(* CODESYS project XtsCore.library
   Version: 0.12.1.34
   Title: XtsCore
   Placeholder: XtsCore
   Company: Beckhoff Automation LLC

Project tree, tasks and I/O mapping:
  libraries: Core, * (Beckhoff Automation LLC); Tc2_Math, * (Beckhoff Automation GmbH); Tc2_MC2, * (Beckhoff Automation GmbH); Tc2_Standard, * (Beckhoff Automation GmbH); Tc2_System, * (Beckhoff Automation GmbH); Tc2_Utilities, * (Beckhoff Automation GmbH); Tc3_EventLogger, * (Beckhoff Automation GmbH); Tc3_McCollisionAvoidance, * (Beckhoff Automation GmbH); Tc3_McCoordinatedMotion, * (Beckhoff Automation GmbH); Tc3_Module, * (Beckhoff Automation GmbH); Tc3_XTS_Utility, * (Beckhoff Automation GmbH)
  _Internal/
    _Needs Sorting/
      global variables TE2000
      function block TE2000_Hmi [ST]: RefreshXtsModule, RefreshXtsMovers, RefreshXtsParts, RefreshXtsPositionTriggers, RefreshXtsStations, RefreshXtsZones, BuildHMI, ControlObject, CyclicLogic, FB_Init, VisitComponent, VisitModule
      global variables TE2000_HMI_Parameters
    Collections/
      Modules/
        ModuleCollection/
          Interfaces/
            interface I_ContainXtsModules: XtsModules
            interface I_XtsModuleCollection: Clear, Count, Create, GetById, GetByOtcid, IsEmpty
            interface I_XtsModuleEnumerator: Current, CurrentItem, MoveToNext, ResetIterator
            function block XtsModuleCollectionAdapter [ST]: AddItem, Clear, Count, Current, CurrentItem, FB_Init, IsEmpty, MoveToNext, RemoveItem, ResetIterator
          function block XtsModuleCollection [ST]: Clear, Count, Create, GetById, GetByOtcid, IsEmpty, Current, CurrentItem, MoveToNext, ResetIterator, Dispose, FB_Exit, AcceptPeeker, CheckModuleId, GetModuleInstance
      Movers/
        MoverCollection/
          Interfaces/
            interface I_XtsMoverCollection: AcceptMoverVisitor, AddItem, Clear, Count, IsEmpty, Remove
            interface I_XtsMoverEnumerator: Current, CurrentItem, MoveToNext, ResetIterator
            interface I_XtsMoverMap: Map
          function block XtsMoverCollection [ST]: Current, CurrentItem, MoveToNext, ResetIterator, AcceptMoverVisitor, AcceptPeeker, AddItem, Clear, Count, IsEmpty, Map, Remove
        MoverList/
          Interfaces/
            interface I_XtsMoverList: Contains, GetAtIndex, InsertAtIndex, RemoveAtIndex
          function block XtsMoverList [ST]: AcceptMoverVisitor, AddItem, Clear, Count, IsEmpty, Map, Remove, Current, CurrentItem, MoveToNext, ResetIterator, Contains, GetAtIndex, InsertAtIndex, Movers, RemoveAtIndex
        MoverQueue/
          Interfaces/
            interface I_XtsMoverQueue: Clear, Count, Dequeue, Enqueue, Peek
          function block XtsMoverQueue [ST]: Current, CurrentItem, Map, MoveToNext, ResetIterator, AcceptMoverVisitor, Clear, Count, Dequeue, Enqueue, Movers, Peek
          function block XtsMoverUniqueQueue [ST]: Enqueue
      Parts/
        PartCollection/
          Interfaces/
            interface I_ContainXtsParts: Parts
            interface I_XtsPartCollection: AddItem, Clear, Count, GetById, GetByOtcid, IsEmpty, Remove
            interface I_XtsPartEnumerator: Current, CurrentItem, MoveToNext, ResetIterator
          function block XtsPartCollection [ST]: Current, CurrentItem, MoveToNext, ResetIterator, AcceptPeeker, AddItem, Clear, Count, FB_Exit, GetById, GetByOtcid, IsEmpty, Remove
      PositionTriggers/
        PositionTriggerCollection/
          Interfaces/
            interface I_XtsPositionTriggerCollection: AddItem, Clear, Count, IsEmpty, Remove
            interface I_XtsPositionTriggerEnumerator: Current, CurrentItem, MoveToNext, ResetIterator
          function block XtsPositionTriggerCollection [ST]: Current, CurrentItem, MoveToNext, ResetIterator, AcceptPeeker, AcceptXtsPositionTriggerVisitor, AddItem, Clear, Count, IsEmpty, Remove
      Stations/
        StationCollection/
          Interfaces/
            interface I_XtsStationCollection: AddItem, Clear, Count, IsEmpty, Remove
            interface I_XtsStationEnumerator: Current, CurrentItem, MoveToNext, ResetIterator
          function block XtsStationCollection [ST]: Current, CurrentItem, MoveToNext, ResetIterator, AcceptPeeker, AcceptStationVisitor, AddItem, Clear, Count, IsEmpty, Remove
      Tracks/
        TrackCollection/
          Interfaces/
            interface I_XtsTrackCollection: Clear, Count, Create, GetById, GetByOtcid, IsEmpty
            interface I_XtsTrackEnumerator: Current, CurrentIndex, MoveToNext, ResetIterator
          function block XtsTrackCollection [ST]: Clear, Count, Create, GetById, GetByOtcid, IsEmpty, Current, CurrentIndex, MoveToNext, ResetIterator, CheckTrackId, GetTrackInstance, FB_Exit
      Zones/
        ZoneCollection/
          Interfaces/
            interface I_XtsZoneCollection: AddItem, Clear, Count, IsEmpty, Remove
            interface I_XtsZoneEnumerator: Current, CurrentItem, MoveToNext, ResetIterator
          function block XtsZoneCollection [ST]: Current, CurrentItem, MoveToNext, ResetIterator, AcceptPeeker, AddItem, Clear, Count, IsEmpty, Remove
      interface I_ContainXtsMoverEnumerator: Movers
      interface I_ContainXtsMoverList: Movers
      interface I_OperatesOnMovers: Movers
    Frames/
      Interfaces/
        interface I_BaseFrame: FrameName
        interface I_FrameModulo: ModuloLength
        interface I_FrameOffset: OffsetToParent
        interface I_HasAReferenceFrame: ReferenceFrame, SetReferenceFrame
        interface I_InGlobalSpace: OffsetToGlobal
        interface I_Positionable: Position
        interface I_ReferencedPosition
        interface I_ReferenceFrame
      function block ReferencedPosition [ST]: Position, ReferenceFrame, SetReferenceFrame
      function block ReferenceFrame [ST]: FB_Init, FrameName, ModuloLength, OffsetToGlobal, OffsetToParent, ReferenceFrame, SetReferenceFrame
    GroupController/
      DUTs/
        data type E_MoverGroupState
      Interfaces/
        interface I_ContainXtsMoverGroupController: XtsMoverGroupController
        interface I_XtsMoverGroupController: AxesGroup, GroupStatus
      function block XtsGroupController [ST]: Disable, Enable, Reset, Accept, AxesGroup, Busy, CyclicLogic, DeregisterWithParent, Done, Enabled, Error, ErrorId, GroupStatus, RegisterWithParent, TaskName
    Module/
      Interfaces/
    Mover/
      MoverTaskBase/
        Interfaces/
          interface I_XtsMoverTask: Axis, Execute
          interface I_XtsMoverTaskCollection: AddTask, ErrorTask, GetTaskById, GetTaskByName, RemoveTaskById, RemoveTaskByInstance
          interface I_XtsMoverTaskResult: Aborted, CommandExecuted, TaskId
        function block XtsMoverTaskCollection [ST]: Busy, Error, ErrorId, ErrorTask, AddTask, CyclicLogic, FB_Init, GetTaskById, GetTaskByName, RemoveTaskById, RemoveTaskByInstance, Reset
        function block XtsMoverTaskResult [ST]: Aborted, CommandExecuted, CyclicLogic, Mover, TaskId
      Parameters/
        Interfaces/
          interface I_BaseDynamics: Acceleration, Deceleration, Direction, Jerk, Velocity
          interface I_CollisionAvoidanceDynamics: Gap
          interface I_CollisionAvoidanceGroupable: AxesGroup, IdentInGroup
          interface I_ContainSyncAxisParameters: SyncAxis
          interface I_HasXtsParameters: Parameters
          interface I_MoveToPositionParameters: Position
          interface I_MoveToStationParameters: Station
          interface I_SyncAxisParameters: MasterAxis, MasterStartDistance, MasterSyncPosition, Options_CA, RatioDenominator, RatioNumerator, SlaveSyncPosition, SyncMode, SyncStrategy
          interface I_XtsParameterSet: CopyFrom, CopyTo
          interface I_XtsTrackParameter: Track
        function block BaseDynamics [ST]: Acceleration, Deceleration, Direction, Jerk, Velocity
        function block CollisionAvoidanceDynamics [ST]: Gap
        function block MoveToPositionParameters [ST]: Position
        function block MoveToStationParameters [ST]: Station
        function block SyncAxisParameters [ST]: MasterAxis, MasterStartDistance, MasterSyncPosition, Options_CA, RatioDenominator, RatioNumerator, SlaveSyncPosition, SyncMode, SyncStrategy
        function block XtsParameterSet [ST]: Acceleration, CopyFrom, CopyTo, Deceleration, Direction, Gap, Jerk, Position, SyncAxis, Track, Velocity
        function block XtsTrackParameter [ST]: Track
      Properties/
        interface I_AxisTrackPositionable: Axis, MoverUtility, PartPosition, Position, TrackPosition
        function block PositionableBehavior [ST]: Axis, CyclicLogic, FB_Init, MoverUtility, PartPosition, Position, TrackPosition
      Status/
        Interfaces/
          interface I_ContainXtsMoverStatus: Status
          interface I_XtsMoverStatus: ActualAcceleration, ActualVelocity, AvoidingCollision, Axis, CommandedPosition, CommandedStation, CurrentTrack, IdentInGroup, InSync, MoverInGroup, SetAcceleration, SetVelocity
        function block XtsMoverStatus [ST]: ActualAcceleration, ActualVelocity, AvoidingCollision, Axis, CommandedPosition, CommandedStation, CurrentTrack, FB_Init, IdentInGroup, InSync, MoverInGroup, SetAcceleration, SetVelocity
      Tasks/
        Interfaces/
          interface I_AxesGroupTask
          interface I_AxisRef: Axis
          interface I_EnableXtsMoverTask: Disable, Disabled, Enable, Enabled, InhibitFeedBackward, InhibitFeedForward, Override
          interface I_MoveToStationTask
          interface I_TakesTrackId: TrackId
        Wrappers/
          Interfaces/
            interface I_ActivateTrack: Execute, TrackId, Busy, Error, ErrorId
            interface I_AxisOnGroup: Execute, IdentInGroup, Busy, Error, ErrorId
            interface I_BaseCollisionAvoidance: Execute, Gap, Active, Busy, Error, ErrorId
            interface I_DynamicsCollisionAvoidance: Acceleration, Deceleration, Jerk, Velocity, CommandAborted
            interface I_GearInPosCA: BufferMode, ContinuousUpdate, MasterStartDistance, MasterSyncPosition, Options, RatioDenominator, RatioNumerator, SlaveSyncPosition, SyncMode, SyncStrategy, InSync, StartSync
            interface I_HaltCa: Deceleration, Jerk, Options, CommandAborted
            interface I_MoveToPositionCA: BufferMode, ContinuousUpdate, Direction, Options, Position, CommandAborted
            interface I_Power: BufferMode, Enable, Enable_Negative, Enable_Positive, Options, Override, Busy, Error, ErrorId, Status
            interface I_ResetAxis: Execute, Busy, Error, ErrorId
          function block ActivateTrack [ST]: Execute, TrackId, Busy, Done, Error, ErrorId
          function block AddAxisToGroup [ST]: Execute, IdentInGroup, Busy, Done, Error, ErrorId
          function block GearInPosCa [ST]: Acceleration, BufferMode, ContinuousUpdate, Deceleration, Execute, Gap, Jerk, MasterStartDistance, MasterSyncPosition, Options, RatioDenominator, RatioNumerator, SlaveSyncPosition, SyncMode, SyncStrategy, Velocity, Active, Busy, CommandAborted, Done, Error, ErrorId, InSync, StartSync
          function block HaltCa [ST]: Deceleration, Execute, Gap, Jerk, Options, Active, Busy, CommandAborted, Done, Error, ErrorId
          function block MoveToAbsolutePositionCA [ST]: Acceleration, BufferMode, ContinuousUpdate, Deceleration, Direction, Execute, Gap, Jerk, Options, Position, Velocity, Active, Busy, CommandAborted, Done, Error, ErrorId
          function block MoveToRelativePositionCA [ST]: Acceleration, BufferMode, ContinuousUpdate, Deceleration, Direction, Execute, Gap, Jerk, Options, Position, Velocity, Active, Busy, CommandAborted, Done, Error, ErrorId
          function block PowerAxis [ST]: BufferMode, Enable, Enable_Negative, Enable_Positive, Options, Override, Busy, Error, ErrorId, Status
          function block RemoveAxisFromGroup [ST]: Execute, IdentInGroup, Busy, Done, Error, ErrorId
          function block ResetMover [ST]: Execute, Busy, Done, Error, ErrorId
        function block _DefaultMoverTasks [ST]
        function block _MoverTasks [ST]: ActivateTrack, AddToGroup, EnableAxis, HaltMover, MoveRelative, MoveToPosition, MoveToStation, MoveVelocity, RemoveFromGroup, ResetAxis, ResetToDefault, SyncToAxis
        function block ActivateTrackTask [ST]: Axis, CyclicLogic, Execute, FB_Init, Reset, TrackId
        function block AddToGroupTask [ST]: AxesGroup, Axis, CyclicLogic, Execute, FB_Init, IdentInGroup, Reset
        function block EnableAxisTask [ST]: Axis, CyclicLogic, Disable, Disabled, Enable, Enabled, Execute, FB_Init, InhibitFeedBackward, InhibitFeedForward, Override, Reset
        function block HaltMoverCATask [ST]: Axis, CyclicLogic, Execute, FB_Init, Interrupted, Reset
        function block MoveRelativeCATask [ST]: Axis, CyclicLogic, Execute, FB_Init, Reset
        data type MoverTaskID
        function block MoveToPositionCATask [ST]: Axis, CyclicLogic, Execute, FB_Init, Reset
        function block MoveToStationTask [ST]: Axis, CyclicLogic, Execute, FB_Init, Reset, Station
        function block MoveVelocityTask [ST]: Axis, CyclicLogic, Execute, FB_Init, Reset
        function block RemoveFromGroupTask [ST]: AxesGroup, Axis, CyclicLogic, Execute, FB_Init, IdentInGroup, Reset
        function block ResetAxisTask [ST]: Axis, CyclicLogic, Execute, FB_Init, Reset
        function block SyncToAxisTask [ST]: Axis, CyclicLogic, Execute, FB_Init, Reset
    NullObjects/
      function GetSeverityString [ST]
      interface I_NullObject
      function block NullAxisRef [ST]: Axis
      function block NullMechatronicsLocalLog [ST]: Clear, Commands, DetailedCommands
      function block NullMechatronicsLogger [ST]: LogMessage, LogMessageInstance
      function block NullMechatronicsTracePublisher [ST]: LogMessage, LogMessageInstance, Subscribe, Unsubscribe
      function block NullMoverCollection [ST]: AcceptMoverVisitor, AddItem, Clear, Count, Current, CurrentItem, IsEmpty, Map, MoveToNext, Remove, ResetIterator
      global variables NullObjects
      function block NullPositionTriggerCollection [ST]: AcceptXtsPositionTriggerVisitor, AddItem, Clear, Count, Current, CurrentItem, IsEmpty, MoveToNext, Remove, ResetIterator
      function block NullReferenceFrame [ST]: FrameName, ModuloLength, OffsetToGlobal, OffsetToParent, ReferenceFrame, SetReferenceFrame
      function block NullStation [ST]: AcceptStationVisitor, CommandLog, CyclicLogic, DeregisterMover, Disable, Enable, Enabled, GetMover, IsMoverRegistered, MoverIsPresent, Movers, Position, RegisterMover, Status, TracePublisher
      function block NullStationCollection [ST]: AcceptStationVisitor, AddItem, Clear, Count, Current, CurrentItem, IsEmpty, MoveToNext, Remove, ResetIterator
      function block NullSyncAxisParameters [ST]: MasterAxis, MasterStartDistance, MasterSyncPosition, Options_CA, RatioDenominator, RatioNumerator, SlaveSyncPosition, SyncMode, SyncStrategy
      function block NullXtsModule [ST]: Accept, AcceptXtsModuleVisitor, CurveAngle, CyclicLogic, Dispose, Gap, HMI, Id, Initialize, Initialized, Length, Module24Vdc, Module48Vdc, ModuleReady, Name, Otcid, RegisterWithParent, Utility, Vdc24Okay, Vdc48Okay, XtsModuleType
      function block NullXtsModuleCollection [ST]: Clear, Count, Create, Current, CurrentItem, Dispose, GetById, GetByOtcid, IsEmpty, MoveToNext, ResetIterator
      function block NullXtsMover [ST]: Accept, AcceptMoverVisitor, ActivateTrack, AddToGroup, Axis, Busy, CommandLog, CurrentTask, DeregisterWithParent, Disable, Enable, Enabled, Error, ErrorId, Halt, Initialize, Initialized, InPosition, InVelocity, LastCyclePosition, ManualGroupControl, MoverData, MoveRelative, MoverId, MoverTasks, MoverUtility, MoveToPosition, MoveToPositionRelative, MoveToStation, MoveVelocity, Name, Parameters, Position, RefreshMoverId, RegisterWithParent, RemoveFromGroup, Reset, Status, SyncToAxis, SyncToMover, TracePublisher, Tracks, VirtualMover
      function block NullXtsMoverData [ST]
      function block NullXtsMoverList [ST]: AcceptMoverVisitor, AddItem, Clear, Contains, Count, Current, CurrentItem, GetAtIndex, InsertAtIndex, IsEmpty, Map, Mover, MoveToNext, Remove, RemoveAtIndex, ResetIterator
      function block NullXtsMoverStatus [ST]: ActualAcceleration, ActualVelocity, AvoidingCollision, Axis, CommandedPosition, CommandedStation, CurrentStation, CurrentTrack, IdentInGroup, InSync, MoverInGroup, SetAcceleration, SetVelocity
      function block NullXtsMoverTask [ST]: Axis, CyclicLogic, Execute, Reset, TaskId, TaskName
      function block NullXtsMoverTaskCollection [ST]: AddTask, ErrorTask, GetTaskById, GetTaskByName, RemoveTaskById, RemoveTaskByInstance
      function block NullXtsMoverTaskResult [ST]: Aborted, Busy, CommandExecuted, Error, ErrorId, TaskId, TaskName
      function block NullXtsParameterSet [ST]: Acceleration, CopyFrom, CopyTo, Deceleration, Direction, Gap, Jerk, Position, SyncAxis, Track, Velocity
      function block NullXtsPart [ST]: Accept, AcceptXtsModuleVisitor, AcceptXtsPartVisitor, Components, CyclicLogic, DeregisterComponent, DeregisterCyclic, DeregisterInitialize, DeregisterModule, DeregisterWithParent, Dispose, Id, Initialize, Initialized, Modules, Name, NumberModulesNotReady, NumberModulesReady, PartReady, Properties, RegisterComponent, RegisterCyclic, RegisterInitialize, RegisterModule, RegisterWithParent, ResetComponents, ResetModules, Utility, Vdc24Okay, Vdc48Okay, XtsModules, XtsPartId
      function block NullXtsPartCollection [ST]: AddItem, Clear, Count, Current, CurrentItem, GetById, GetByOtcid, IsEmpty, MoveToNext, Remove, ResetIterator
      function block NullXtsPartTask [ST]: Busy, Error, ErrorId, TaskName, XtsPartId
      function block NullXtsPositionTrigger [ST]: Accept, AcceptXtsPositionTriggerVisitor, CommandLog, DeregisterMover, DeregisterWithParent, Disable, Enable, Enabled, GetMover, IsMoverRegistered, MoverIsPresent, MoverQueue, Movers, Name, Position, RegisterMover, RegisterWithParent, Status, TracePublisher
      function block NullXtsPositionTriggerStatus [ST]: NumberOfMoverEvents, NumberOfMoversRegistered
      function block NullXtsStationStatus [ST]: CurrentMoverId, CurrentMoverName, NumberOfMoversRegistered
      function block NullXtsSystem [ST]: Accept, AcceptMoverVisitor, AcceptStationVisitor, AcceptXtsModuleVisitor, AcceptXtsPartVisitor, AcceptXtsPositionTriggerVisitor, AcceptXtsZoneVisitor, AxesGroupRef, Busy, CAGroupErrorId, CaGroupStatus, CommandLog, Components, Config, CurrentTask, CyclicLogic, DeregisterComponent, DeregisterCyclic, DeregisterInitialize, DeregisterModule, DeregisterWithParent, Disable, DisableGroup, DisableMovers, Enable, Enabled, EnableGroup, EnableMovers, Environment, Error, ErrorId, Initialize, Initialized, ManualDiagnoser, Modules, Movers, MoversEnabled, Name, Parameters, Parts, PositionTriggers, RegisterComponent, RegisterCyclic, RegisterInitialize, RegisterModule, RegisterWithParent, Reset, ResetCaGroup, ResetComponents, ResetModules, ResetMovers, RetriggerMoverDetection, Stations, Status, TracePublisher, Tracks, TriggerMoverDetection, TriggerMoverIdentification, Utility, UtilityProperties, XpuId, XtsTasks, Zones
      function block NullXtsSystemConfiguration [ST]: CommandPositionTriggersOnDisable, CommandPositionTriggersOnEnable, CommandStationsOnDisable, CommandStationsOnEnable
      function block NullXtsSystemStatus [ST]: CyclicLogic, NumberOfMovers, NumberOfParts, NumberOfPositionTriggers, NumberOfStations, NumberOfTracks, NumberOfZones, NumberPartsNotReady, NumberPartsReady, Simulated, Vdc24Okay, Vdc48Okay
      function block NullXtsSystemTasks [ST]: AddTask, CyclicLogic, GetTaskById, GetTaskByName, RemoveTaskById, RemoveTaskByInstance
      function block NullXtsTask [ST]: Busy, Error, ErrorId, TaskId, TaskName, XpuId
      function block NullXtsTrack [ST]: Dispose, Id, Length, Offset, Otcid, Polarity, Utility
      function block NullXtsTrackCollection [ST]: Clear, Count, Create, Current, CurrentIndex, GetById, GetByOtcid, IsEmpty, MoveToNext, ResetIterator
      function block NullXtsZone [ST]: Accept, AcceptMoverVisitor, AcceptXtsZoneVisitor, CommandLog, DeregisterWithParent, EndPosition, GetSortedMover, IsMoverInZone, Length, MonitoredMovers, Movers, Name, RegisterWithParent, StartPosition, Status, TracePublisher
      function block NullXtsZoneStatus [ST]: NumberOfMoversInZone
      function block NullZoneCollection [ST]: AddItem, Clear, Count, Current, CurrentItem, IsEmpty, MoveToNext, Remove, ResetIterator
    Parts/
      Properties/
        interface I_ContainXtsPartProperties: Properties
        interface I_XtsPartProperties: General
        interface I_XtsPartPropertiesGeneral: ModuleSide, Offset, OTCID
        function block XtsPartProperties [ST]: General
        function block XtsPartPropertiesGeneral [ST]: ModuleSide, Offset, OTCID
      Tasks/
        Interfaces/
          interface I_XtsPartInitializeTask
          interface I_XtsPartTask: XtsPartId
          interface I_XtsPartTaskResult
        function block InitializeXtsPartTask [ST]: Initialize, Initialized, XtsPartId
      interface I_XtsPartId: XtsPartId
    Peeker/
      Interfaces/
        interface I_XtsModuleCollectionPeeker: SetCollection
        interface I_XtsMoverCollectionPeeker: SetCollection
        interface I_XtsPartCollectionPeeker: SetCollection
        interface I_XtsPositionTriggerCollectionPeeker: SetCollection
        interface I_XtsStationCollectionPeeker: SetCollection
        interface I_XtsZoneCollectionPeeker: SetCollection
    PositionTrigger/
      Status/
        Interfaces/
          interface I_ContainXtsPositionTriggerStatus: Status
          interface I_XtsPositionTriggerStatus: NumberOfMoverEvents, NumberOfMoversRegistered
        function block XtsPositionTriggerStatus [ST]: FB_Init, NumberOfMoverEvents, NumberOfMoversRegistered, SetRegisteredMovers
    Station/
      DUT/
        data type E_ThresholdEvent
      Interfaces/
        interface I_MoverMonitor: GetMover, MonitoredMovers, MoverPresent
        interface I_StationTaskCollection
      Status/
        Interfaces/
          interface I_ContainXtsStationStatus: Status
          interface I_XtsStationStatus: NumberOfMoversRegistered
        function block XtsStationStatus [ST]: FB_Init, NumberOfMoversRegistered, SetRegisteredMovers
      function CheckForThresholdEvent [ST]
      function block MoverMonitorTask [ST]: CyclicLogic, FB_Init, GetMover, MonitoredMovers, MoverPresent
      function block MoverThresholdMonitorTask [ST]: CyclicLogic, FB_Init, GetMover, MonitoredMovers, MoverPresent, SetMonitoredMovers
    TaskBase/
      Interfaces/
        interface I_TaskResult: TaskName
      function block BaseTaskResult [ST]: Busy, Error, ErrorId, TaskName
    Tracing/
      function block XtsCoreEventLogger [ST]: LogMessage, LogMessageInstance
    Tracks/
      Interfaces/
        interface I_XtsTrack: Id, Length, Offset, Otcid, Polarity, Utility
      function block XtsTrack [ST]: Dispose, Id, Length, Offset, Otcid, Polarity, Utility
    XtsSystem/
      Base/
        Interfaces/
          interface I_XtsTask: XpuId
          interface I_XtsTaskCollection: AddTask, GetTaskById, GetTaskByName, RemoveTaskById, RemoveTaskByInstance
          interface I_XtsTaskResult: TaskId
        function block XtsTaskCollection [ST]: AddTask, Busy, CyclicLogic, Error, ErrorId, FB_Init, GetTaskById, GetTaskByName, RemoveTaskById, RemoveTaskByInstance, Reset
        function block XtsTaskResult [ST]: TaskId
      Properties/
        Interfaces/
          interface I_ContainXtsSystemProperties: UtilityProperties
          interface I_XtsSystemUtilityProperties: Mover
          interface I_XtsSystemUtilityPropertiesMover: XtsMagnetPlateType, XtsMoverType
        function block XtsSystemConfiguration [ST]: CommandPositionTriggersOnDisable, CommandPositionTriggersOnEnable, CommandStationsOnDisable, CommandStationsOnEnable
        function block XtsSystemUtilityProperties [ST]: Mover
        function block XtsSystemUtilityPropertiesMover [ST]: XtsMagnetPlateType, XtsMoverType
      Status/
        Interfaces/
          interface I_ContainXtsSystemStatus: Status
          interface I_XtsSystemStatus: NumberOfMovers, NumberOfParts, NumberOfPositionTriggers, NumberOfStations, NumberOfTracks, NumberOfZones, NumberPartsNotReady, NumberPartsReady, Simulated, Vdc24Okay, Vdc48Okay
        function block XtsSystemStatus [ST]: CyclicLogic, FB_Init, NumberOfMovers, NumberOfParts, NumberOfPositionTriggers, NumberOfStations, NumberOfTracks, NumberOfZones, NumberPartsNotReady, NumberPartsReady, Simulated, Vdc24Okay, Vdc48Okay
      Tasks/
        Interfaces/
          interface I_XtsDisableTask: AxesGroup
          interface I_XtsEnableTask: AxesGroup
          interface I_XtsExecutableTask: Execute
          interface I_XtsInitializeTask
          interface I_XtsMoverDetectionTask
          interface I_XtsMoverIdentificationTask
          interface I_XtsMoverRedetectionTask
        function block _DefaultXtsTasks [ST]
        function block _XtsTasks [ST]: DisableXtsTask, EnableXtsTask, InitializeXtsTask, MoverDetectionTask, MoverIdentificationTask, MoverRedetectionTask
        function block DisableXtsTask [ST]: AxesGroup, CyclicLogic, Execute, FB_Init, Reset, XpuId, XtsMoverCommander, XtsMoverGroupController
        function block EnableXtsTask [ST]: AxesGroup, CyclicLogic, Execute, FB_Init, Reset, XpuId, XtsMoverCommander, XtsMoverGroupController
        function block InitializeXtsTask [ST]: Initialize, Initialized, InfoServerSetup, MoverSetup, PartSetup, TrackSetup, FB_Init, Reset, XpuId
        function block MoverDetectionTask [ST]: Execute, FB_Init, XpuId
        function block MoverIdentificationTask [ST]: CyclicLogic, Execute, FB_Init, Reset, XpuId
        function block MoverRedetectionTask [ST]: Execute, FB_Init, XpuId
        data type XtsSystemTaskId
      function block ManualDebugger [ST]: PartIdForModules, RefreshCollections, SetCollections
    Zone/
      Interfaces/
        interface I_MoverInPositionChecker: IsMoverInPosition
        interface I_XtsMoverComparer: Compare
        interface I_ZoneMonitor
      Properties/
        Interfaces/
          interface I_SingleDimensionZone: EndPosition, StartPosition
        function block _DefaultZoneProperties [ST]
        function block _DefaultZonePropertyBackers [ST]: SingleDimensionBacker
        function block SingleDimensionZone [ST]: EndPosition, StartPosition
      Status/
        Interfaces/
          interface I_ContainXtsZoneStatus: Status
          interface I_XtsZoneStatus: NumberOfMoversInZone
        function block XtsZoneStatus [ST]: FB_Init, NumberOfMoversInZone, SetMoverCollection
      function MoverDistance [ST]
      function block MoverZoneDistanceComparer [ST]: Compare, FB_Init
      function block SingleDimensionChecker [ST]: FB_Init, IsMoverInPosition
      function block ZoneMonitor [ST]: CyclicLogic, FB_Init, MonitoredMovers, Movers
    data type E_XtsLogMessage
  HMI/
    DUT/
      data type ST_LocalLogbook_HMI
      data type ST_MoverCommands_HMI
      data type ST_XtsModule_HMI
      data type ST_XtsMover_HMI
      data type ST_XtsMover_Parameters_HMI
      data type ST_XtsPart_HMI
      data type ST_XtsPartHmiHelper
      data type ST_XtsPositionTrigger_HMI
      data type ST_XtsStation_HMI
      data type ST_XtsSystem_HMI
      data type ST_XtsTrack_HMI
      data type ST_XtsZone_HMI
    function block XtsBasicHmi [ST]: FB_Init, Accept, BuildHMI, ControlObject, CyclicLogic, VisitComponent, VisitModule
    function block XtsModule_HMI [ST]: ControlObject, CyclicLogic, FB_Init, XtsModule
    function block XtsMover_HMI [ST]: ControlObject, CyclicLogic, FB_Init, XtsMover
    function block XtsPart_HMI [ST]: ControlObject, CyclicLogic, FB_Init, XtsPart
    function block XtsPositionTrigger_HMI [ST]: ControlObject, CyclicLogic, FB_Init, XtsPositionTrigger
    function block XtsStation_HMI [ST]: ControlObject, CyclicLogic, FB_Init, XtsStation
    function block XtsSystem_HMI [ST]: ControlObject, CyclicLogic, FB_Init
    function block XtsZone_HMI [ST]: ControlObject, CyclicLogic, FB_Init
  Logging/
    Interfaces/
      interface I_ContainXtsLocalLog: CommandLog
      interface I_ContainXtsTracePublisher: TracePublisher
      interface I_XtsLocalLog: Clear, Commands, DetailedCommands
      interface I_XtsLocalLogger
      interface I_XtsLogCommand
      interface I_XtsLogger
      interface I_XtsTracePublisher: Subscribe, Unsubscribe
    function block XtsLocalLogger [ST]: Clear, Commands, DetailedCommands, FB_Init, LogMessage, LogMessageInstance
    function block XtsLogCommand [ST]: Arguments, Message, MessageId, Severity, SourceId, SourceName, TimeStamp
    function block XtsTracePublisher [ST]: LogMessage, LogMessageInstance, Subscribe, Unsubscribe
  MoverVisitors/
    Interfaces/
      interface I_XtsMoverVisitorTask: ExecuteOn
    MoverCollectionVisitors/
    function block XtsMoverActivateTrack [ST]: CopyParametersFrom, TrackId, XtsMoverVisitee, Aborted, Busy, CommandExecuted, Error, ErrorId, ExecuteOn, TaskId, TaskName, VisitMover
    function block XtsMoverAddToGroup [ST]: AxesGroup, IdentInGroup, XtsMoverVisitee, Aborted, Busy, CommandExecuted, Error, ErrorId, ExecuteOn, TaskId, TaskName, VisitMover
    function block XtsMoverDisabler [ST]: XtsMoverVisitee, Aborted, Busy, CommandExecuted, Error, ErrorId, ExecuteOn, TaskId, TaskName, VisitMover
    function block XtsMoverEnabler [ST]: XtsMoverVisitee, Aborted, Busy, CommandExecuted, Error, ErrorId, ExecuteOn, TaskId, TaskName, VisitMover
    function block XtsMoverHalt [ST]: CopyParametersFrom, Deceleration, Gap, Jerk, XtsMoverVisitee, Aborted, Busy, CommandExecuted, Error, ErrorId, ExecuteOn, TaskId, TaskName, VisitMover
    function block XtsMoverMoveToPosition [ST]: Acceleration, CopyParametersFrom, Deceleration, Direction, Gap, Jerk, Position, Velocity, XtsMoverVisitee, Aborted, Busy, CommandExecuted, Error, ErrorId, ExecuteOn, TaskId, TaskName, VisitMover
    function block XtsMoverMoveToStation [ST]: Acceleration, CopyParametersFrom, Deceleration, Direction, Gap, Jerk, Station, Velocity, XtsMoverVisitee, Aborted, Busy, CommandExecuted, Error, ErrorId, ExecuteOn, TaskId, TaskName, VisitMover
    function block XtsMoverMoveVelocity [ST]: Acceleration, CopyParametersFrom, Deceleration, Direction, Gap, Jerk, Velocity, XtsMoverVisitee, Aborted, Busy, CommandExecuted, Error, ErrorId, ExecuteOn, TaskId, TaskName, VisitMover
    function block XtsMoverRemoveFromGroup [ST]: AxesGroup, IdentInGroup, XtsMoverVisitee, Aborted, Busy, CommandExecuted, Error, ErrorId, ExecuteOn, TaskId, TaskName, VisitMover
  Project Information/
    function F_GetCompany [ST]
    function F_GetTitle [ST]
    function F_GetVersion [ST]
  Utilities/
    Logging/
      global variables XtsTrace
    Validators/
      function block AllMoversValidator [ST]: Valid
      function block NoMoversValidator [ST]: Valid
    function IsNullObject [ST]
    function IsValidObject [ST]
  Version/
    global variables Global_Version
  XtsModule/
    Interfaces/
      interface I_AcceptXtsModuleVisitor: AcceptXtsModuleVisitor
      interface I_ContainXtsPartModuleUtility: Utility
      interface I_XtsModule: CurveAngle, Gap, Id, Length, ModuleReady, Otcid, Vdc24Okay, Vdc48Okay, XtsModuleType
      interface I_XtsModuleVisitor: VisitXtsModule
    function block XtsModule [ST]: DeregisterWithParent, RegisterWithParent, Dispose, Initialize, Initialized, CurveAngle, Gap, Id, Length, ModuleReady, Otcid, Utility, Vdc24Okay, Vdc48Okay, XtsModuleType, AcceptXtsModuleVisitor, CyclicLogic
  XtsMover/
    Interfaces/
      interface I_AcceptXtsMoverVisitors: AcceptMoverVisitor
      interface I_XtsCommands: ActivateTrack, AddToGroup, Halt, MoveRelative, MoveToPosition, MoveToStation, MoveVelocity, RemoveFromGroup, SyncToAxis, SyncToMover
      interface I_XtsMover: CurrentTask, InPosition, InVelocity, LastCyclePosition, ManualGroupControl, MoverId, MoverTasks, Position, RefreshMoverId, Tracks, VirtualMover
      interface I_XtsMoverUtility: MoverUtility
      interface I_XtsMoverValidator: Valid
      interface I_XtsMoverVisitor: VisitMover
    XtsMoverData/
      Interfaces/
        interface I_ContainXtsMoverData: MoverData
        interface I_XtsMoverData
    function block XtsMover [ST]: CyclicLogic, MoverTasks, MoverUtility, RefreshMoverId, RegisterWithParent, ActivateTrack, AddToGroup, Disable, Enable, Halt, MoveRelative, MoveToPosition, MoveToStation, MoveVelocity, RemoveFromGroup, Reset, SyncToAxis, SyncToMover, FB_Init, Initialize, Initialized, Axis, InhibitFeedBackward, InhibitFeedForward, InPosition, InVelocity, LastCyclePosition, ManualGroupControl, MoverData, MoverId, Override, Parameters, Position, Tracks, VirtualMover, Busy, CurrentTask, Enabled, Error, ErrorId, Status, CommandLog, TracePublisher, AcceptMoverVisitor
  XtsMoverCommander/
    Interfaces/
      interface I_ContainXtsMoverCommander: XtsMoverCommander
      interface I_XtsMoverCommander: ActivateTrack, AddToGroup, Disable, Enable, Halt, MoveToPosition, MoveToStation, MoveVelocity, RemoveFromGroup
    function block XtsMoverCommander [ST]: ActivateTrack, AddToGroup, Disable, Enable, Halt, MoveToPosition, MoveToStation, MoveVelocity, RemoveFromGroup, Busy, CurrentTask, Error, ErrorId, Parameters, TaskName
  XtsPart/
    Interfaces/
      interface I_AcceptXtsPartVisitor: AcceptXtsPartVisitor
      interface I_ContainXtsPartUtility: Utility
      interface I_XtsPart: PartReady, Vdc24Okay, Vdc48Okay
      interface I_XtsPartVisitor: VisitXtsPart
    function block XtsPart [ST]: FB_Init, Dispose, Initializing, Properties, PartReady, Vdc24Okay, Vdc48Okay, AcceptXtsModuleVisitor, AcceptXtsPartVisitor, OnCyclicCall, Utility, XtsModules, XtsPartId
  XtsPositionTrigger/
    Interfaces/
      interface I_AcceptXtsPositionTriggerVisitor: AcceptXtsPositionTriggerVisitor
      interface I_Queueable: MoverQueue
      interface I_VisitXtsPositionTrigger: VisitXtsPositionTrigger
      interface I_XtsPositionTrigger: Movers
    function block XtsPositionTrigger [ST]: FB_Init, Disable, Enable, Enabled, CommandLog, TracePublisher, AcceptXtsPositionTriggerVisitor, CyclicLogic, DeregisterMover, GetMover, IsMoverRegistered, MoverIsPresent, MoverQueue, Movers, Position, RegisterMover, Status
  XtsStation/
    Interfaces/
      interface I_AcceptXtsStationVisitor: AcceptStationVisitor
      interface I_MoverPositionMonitor
      interface I_Station: DeregisterMover, GetMover, IsMoverRegistered, MoverIsPresent, RegisterMover
      interface I_XtsStation
      interface I_XtsStationVisitor: VisitStation
    function block XtsStation [ST]: FB_Init, Disable, Enable, Enabled, CommandLog, TracePublisher, AcceptStationVisitor, CyclicLogic, DeregisterMover, GetMover, IsMoverRegistered, MoverIsPresent, Movers, Position, RegisterMover, Status
  XtsSystem/
    Interfaces/
      interface I_ContainXtsEnvironment: Environment
      interface I_ContainXtsMovers: Movers
      interface I_ContainXtsPositionTriggers: PositionTriggers
      interface I_ContainXtsStations: Stations
      interface I_ContainXtsTracks: Tracks
      interface I_ContainXtsUtility: Utility
      interface I_ContainXtsZones: Zones
      interface I_XtsSystem: AxesGroupRef, Busy, CAGroupErrorId, CaGroupStatus, Config, CurrentTask, Error, ErrorId, ManualDiagnoser, MoversEnabled, XtsTasks
      interface I_XtsSystemCommands: DisableGroup, DisableMovers, EnableGroup, EnableMovers, ResetCaGroup, ResetMovers, RetriggerMoverDetection, TriggerMoverDetection, TriggerMoverIdentification
      interface I_XtsSystemConfiguration: CommandPositionTriggersOnDisable, CommandPositionTriggersOnEnable, CommandStationsOnDisable, CommandStationsOnEnable
      interface I_XtsXpuId: XpuId
    function block XtsSystem [ST]: Movers, Parameters, Parts, PositionTriggers, Stations, Tracks, XtsTasks, Zones, Disable, DisableGroup, DisableMovers, Enable, EnableGroup, EnableMovers, Reset, ResetCaGroup, ResetMovers, RetriggerMoverDetection, TriggerMoverDetection, TriggerMoverIdentification, FB_Init, Initializing, UtilityProperties, AxesGroupRef, Busy, CAGroupErrorId, CaGroupStatus, Config, CurrentTask, Enabled, Environment, Error, ErrorId, MoversEnabled, Status, Utility, XpuId, CommandLog, TracePublisher, AcceptMoverVisitor, AcceptStationVisitor, AcceptXtsModuleVisitor, AcceptXtsPartVisitor, AcceptXtsPositionTriggerVisitor, AcceptXtsZoneVisitor, ManualDiagnoser, OnCyclicCall
  XtsZone/
    Interfaces/
      interface I_AcceptXtsZoneVisitor: AcceptXtsZoneVisitor
      interface I_MonitorsMovers: MonitoredMovers
      interface I_XtsZone: GetSortedMover, IsMoverInZone
      interface I_XtsZoneVisitor: VisitZone
    function block XtsZone [ST]: FB_Init, EndPosition, StartPosition, CommandLog, TracePublisher, AcceptMoverVisitor, AcceptXtsZoneVisitor, CyclicLogic, GetSortedMover, IsMoverInZone, MonitoredMovers, Movers, Status
  global variables XtsCoreParameters
*)

// _Internal/GroupController/DUTs/E_MoverGroupState
{attribute 'qualified_only'}
{attribute 'strict'}
{attribute 'to_string'}
TYPE E_MoverGroupState :
(
	Disabled := 0,
	NotReady,
	Standby,
	Moving,
	Stopping,
	Error
);
END_TYPE

// _Internal/Mover/Tasks/MoverTaskID
{attribute 'qualified_only'}
{attribute 'strict'}
{attribute 'to_string'}
TYPE MoverTaskID : 
(
	ENABLE,
	DISABLE,
	MOVE_TO_POSITION,
	MOVE_RELATIVE,
	MOVE_TO_STATION,
	MOVE_VELOCITY,
	HALT_MOVER,
	ADD_TO_GROUP,
	REMOVE_FROM_GROUP,
	ACTIVATE_TRACK,
	RESET_MOVER,	
	SYNC_TO_AXIS,
	NCT,
	CUSTOM_1,
	CUSTOM_2
) UDINT;
END_TYPE

// _Internal/Station/DUT/E_ThresholdEvent
{attribute 'qualified_only'}
{attribute 'strict'}
{attribute 'to_string'}
TYPE E_ThresholdEvent : (
		NoEvent		  := 0,
		PositiveEvent := 1,
		NegativeEvent := 2
	);
END_TYPE

// _Internal/XtsSystem/Tasks/XtsSystemTaskId
{attribute 'qualified_only'}
{attribute 'to_string'}
TYPE XtsSystemTaskId :
(
	INITIALIZE,
	ENABLE,
	DISABLE,
	MOVER_DETECTION,
	MOVER_REDETECTION,
	MOVER_IDENTIFICATION,
	NCT_MANAGER,
	CUSTOM_1,
	CUSTOM_2,
	CUSTOM_3	
) UDINT;
END_TYPE

// _Internal/E_XtsLogMessage
{attribute 'qualified_only'}
{attribute 'strict'}
{attribute 'to_string'}
TYPE E_XtsLogMessage : (
		SystemVerbose								:= 0,
		SystemInfo									:= 1,
		SystemWarning								:= 2,
		SystemError									:= 3,
		SystemCriticalError							:= 4,
		SystemInitializationStarted					:= 20,
		SystemInitializationFinished				:= 21,
		SystemInitializationAxesGroupNotLinked		:= 22,
		SystemInitializationAxesGroupLengthMismatch := 23,
		SystemInitializationXpuNameNotFound			:= 24,
		SystemInitializationAxesGroupNotFound		:= 25,
		SystemTrackInitializationStarted			:= 30,
		SystemTrackInitializationFinished			:= 31,
		SystemMoverInitializationStarted			:= 32,
		SystemMoverInitializationFinished			:= 33,
		SystemPartInitializationStarted				:= 34,
		SystemPartInitializationFinished			:= 35,
		SystemPartModulesInitializationStarted		:= 36,
		SystemPartModulesInitializationFinished		:= 37,
		SystemEnableActivateTrackFailed				:= 40,
		SystemEnableStationSkipped					:= 41,
		SystemEnablePositionTriggerSkipped			:= 42,
		SystemDisableStationSkipped					:= 43,
		SystemDisablePositionTriggerSkipped			:= 44,
		SystemEnableVoltageCheckFailed				:= 45,
		MoverCommandedToEnable						:= 100,
		MoverCommandedToDisable						:= 101,
		MoverCommandedToStation						:= 102,
		MoverCommandedToPosition					:= 103,
		MoverCommandedToMoveVelocity				:= 104,
		MoverCommandedToAddToGroup					:= 105,
		MoverCommandedToRemoveFromGroup				:= 106,
		MoverCommandedToActivateTrack				:= 107,
		MoverCommandedToHalt						:= 108,
		MoverCommandedToReset						:= 109,
		MoverCommandedToSyncAxis					:= 110,
		MoverCommandedToSyncMover					:= 111,
		MoverCommandErrorInvalidParameter			:= 120,
		MoverCommandGeneralTaskError				:= 121,
		MoverInitializeAxisNotLinked				:= 130,
		MoverRefreshMoverIdInvalidXpu				:= 131,
		MoverRefreshMoverIdNoAxisObjectFound		:= 132,
		StationEnabled								:= 200,
		StationDisabled								:= 201,
		StationMoverRegistered						:= 202,
		StationMoverDeregistered					:= 203,
		StationMoverArrived							:= 204,
		StationGetMoverCalled						:= 205,
		StationGetMoverCalledNoMover				:= 206,
		PositionTriggerEnabled						:= 250,
		PositionTriggerDisabled						:= 251,
		PositionTriggerMoverRegistered				:= 252,
		PositionTriggerMoverDeregistered			:= 253,
		PositionTriggerMoverPassedPositive			:= 254,
		PositionTriggerMoverPassedNegative			:= 255,
		PositionTriggerGetMoverCalled				:= 256,
		ZoneMoverEntered							:= 300,
		ZoneMoverExited								:= 301,
		ZoneMoverErrorTrackLengthZero				:= 302,
		ZoneMoverErrorGetSortedIndexOOB				:= 303
	) UDINT;
END_TYPE

// HMI/DUT/ST_LocalLogbook_HMI
TYPE ST_LocalLogbook_HMI :
	STRUCT
		Logs	 : ARRAY[1..XtsCoreParameters.MaxNumberLocalLog] OF T_MaxString;
		ClearLog : BOOL;
	END_STRUCT
END_TYPE

// HMI/DUT/ST_MoverCommands_HMI
TYPE ST_MoverCommands_HMI :
	STRUCT
		Enable		   : Button;
		Disable		   : Button;
		Reset		   : Button;
		MoveToPosition : Button;
		MoveVelocity   : Button;
		MoveToStation  : Button;
		BumpCommand	   : Button;
		Halt		   : Button;
	END_STRUCT
END_TYPE

// HMI/DUT/ST_XtsModule_HMI
TYPE ST_XtsModule_HMI :
	STRUCT
		Name		: T_MaxString;
		Length		: LREAL;
		CurveAngle	: LREAL;
		Gap			: LREAL;
		ModuleType	: Tc3_Xts_Utility.ModuleType;
		ModuleReady : BOOL;
	END_STRUCT
END_TYPE

// HMI/DUT/ST_XtsMover_HMI
TYPE ST_XtsMover_HMI EXTENDS ST_HmiFunction :
	STRUCT
		Position			 : LREAL;
		Velocity			 : LREAL;
		Acceleration		 : LREAL;
		Deceleration		 : LREAL;
		Jerk				 : LREAL;
		Gap					 : LREAL;
		CurrentTask			 : T_MaxString;
		AvoidingCollision	 : BOOL;
		Commands			 : ST_MoverCommands_HMI;
		Parameters			 : ST_XtsMover_Parameters_HMI;
		MoverInGroup		 : BOOL;
		CommandedPosition	 : LREAL;
		CommandedStationName : T_MaxString;
		Enabled				 : BOOL;
		Busy				 : BOOL;
		HasError			 : BOOL;
		Initialized			 : BOOL;
		ErrorId				 : UDINT;
		Id					 : UDINT;
		IdentInGroup		 : UDINT;
		LocalLog			 : ST_LocalLogbook_HMI;
	END_STRUCT
END_TYPE

// HMI/DUT/ST_XtsMover_Parameters_HMI
TYPE ST_XtsMover_Parameters_HMI :
	STRUCT
		Position	 : LREAL;
		Velocity	 : LREAL;
		Acceleration : LREAL;
		Deceleration : LREAL;
		Jerk		 : LREAL;
		Gap			 : LREAL;
		Distance	 : LREAL;
		Direction	 : Tc3_Mc3Definitions.MC_DIRECTION;
		Station		 : T_MaxString;
	END_STRUCT
END_TYPE

// HMI/DUT/ST_XtsPart_HMI
TYPE ST_XtsPart_HMI EXTENDS ST_HmiFunction :
	STRUCT
		Side			: Tc3_Xts_Utility.ModuleSide;
		Modules			: ARRAY[1..TE2000_HMI_Parameters.NUMBER_OF_MODULES] OF St_XtsModule_HMI;
		X				: LREAL;
		Y				: LREAL;
		Angle			: LREAL;
		NumberOfModules : UDINT;
		PartReady		: BOOL;
		Vdc24Okay		: BOOL;
		Vdc48Okay		: BOOL;
		Id				: UDINT;
	END_STRUCT
END_TYPE

// HMI/DUT/ST_XtsPartHmiHelper
TYPE ST_XtsPartHmiHelper :
	STRUCT
		Part	: I_XtsPart;
		Modules : ARRAY[1..TE2000_HMI_Parameters.NUMBER_OF_MODULES] OF I_XtsModule;
	END_STRUCT
END_TYPE

// HMI/DUT/ST_XtsPositionTrigger_HMI
TYPE ST_XtsPositionTrigger_HMI EXTENDS ST_HmiFunction :
	STRUCT
		Enable				   : Button;
		Disable				   : Button;
		ClearQueue			   : Button;
		Enabled				   : BOOL;
		MoverPresent		   : BOOL;
		Position			   : LREAL;
		TargetPosition		   : LREAL;
		SetPosition			   : BOOL;
		NumberMoversRegistered : UDINT;
		NumberEventsInQueue	   : UDINT;
		LocalLog			   : ST_LocalLogbook_HMI;
	END_STRUCT
END_TYPE

// HMI/DUT/ST_XtsStation_HMI
TYPE ST_XtsStation_HMI EXTENDS ST_HmiFunction :
	STRUCT
		Enable				   : Button;
		Disable				   : Button;
		Enabled				   : BOOL;
		MoverPresent		   : BOOL;
		Position			   : LREAL;
		TargetPosition		   : LREAL;
		SetPosition			   : BOOL;
		NumberMoversRegistered : UDINT;
		LocalLog			   : ST_LocalLogbook_HMI;
	END_STRUCT
END_TYPE

// HMI/DUT/ST_XtsSystem_HMI
TYPE ST_XtsSystem_HMI EXTENDS ST_HmiFunction :
	STRUCT
		Enable					 : Button;
		Enabled					 : BOOL;
		Disable					 : Button;
		ErrorId					 : STRING[10];
		HasError				 : BOOL;
		CurrentTask				 : T_MaxString;
		LastTask				 : T_MaxString;
		Initialized				 : BOOL;
		CaGroup					 : T_MaxString;
		MoversEnabled			 : BOOL;
		Reset					 : Button;
		MoverType				 : Tc3_Xts_Utility.MoverType;
		LocalLog				 : ST_LocalLogbook_HMI;
		NumberOfTracks			 : UDINT;
		NumberOfParts			 : UDINT;
		NumberOfMovers			 : UDINT;
		NumberOfPositionTriggers : UDINT;
		NumberOfStations		 : UDINT;
		NumberOfZones			 : UDINT;
		Simulated				 : BOOL;
		Vdc24Okay				 : BOOL;
		Vdc48Okay				 : BOOL;
	END_STRUCT
END_TYPE

// HMI/DUT/ST_XtsTrack_HMI
TYPE ST_XtsTrack_HMI EXTENDS ST_HmiFunction :
	STRUCT
		Position : LREAL;
	END_STRUCT
END_TYPE

// HMI/DUT/ST_XtsZone_HMI
TYPE ST_XtsZone_HMI EXTENDS ST_HmiFunction :
	STRUCT
		StartPosition	   : LREAL;
		EndPosition		   : LREAL;
		Length			   : LREAL;
		NumberMoversInZone : UDINT;
		SortedPosition	   : UDINT;
		SortedDirection	   : Tc3_Mc3Definitions.MC_DIRECTION := Tc3_Mc3Definitions.MC_DIRECTION.mcDirectionPositive;
		MoverCommands	   : ST_MoverCommands_HMI;
		CommandParameters  : ST_XtsMover_Parameters_HMI;
		GetSortedMover	   : Button;
		SortedMover		   : T_MaxString;
		LocalLog		   : ST_LocalLogbook_HMI;
	END_STRUCT
END_TYPE

// _Internal/_Needs Sorting/TE2000
{attribute 'qualified_only'}
VAR_GLOBAL
// 	HMI			  : TE2000_Hmi<TE2000_Hmi_Parameters.NUMBER_OF_MOVERS,
// 	TE2000_Hmi_Parameters.NUMBER_OF_PARTS,
// 	TE2000_Hmi_Parameters.NUMBER_OF_Modules,
// 	TE2000_Hmi_Parameters.NUMBER_OF_STATIONS,
// 	TE2000_Hmi_Parameters.NUMBER_OF_POSITIONTRIGGERS,
// 	TE2000_Hmi_Parameters.NUMBER_OF_ZONES,
// 	TE2000_Hmi_Parameters.NUMBER_OF_TRACKS>('Sandbox HMI');
END_VAR

// _Internal/_Needs Sorting/TE2000_HMI_Parameters
{attribute 'hidden'}
{attribute 'qualified_only'}
VAR_GLOBAL CONSTANT
	NUMBER_OF_MOVERS		   : UDINT := 10;
	NUMBER_OF_PARTS			   : UDINT := 1;
	NUMBER_OF_MODULES		   : UDINT := 30;
	NUMBER_OF_STATIONS		   : UDINT := 5;
	NUMBER_OF_POSITIONTRIGGERS : UDINT := 5;
	NUMBER_OF_ZONES			   : UDINT := 2;
	NUMBER_OF_TRACKS		   : UDINT := 1;
END_VAR

// _Internal/NullObjects/NullObjects
{attribute 'qualified_only'}
VAR_GLOBAL
	MechatronicsLocalLog	   : NullMechatronicsLocalLog;
	MechatronicsLogger		   : NullMechatronicsLogger;
	MechatronicsTracePublisher : NullMechatronicsTracePublisher;
	MoverCollection			   : NullMoverCollection;
	PositionTriggerCollection  : NullPositionTriggerCollection;
	ReferenceFrame			   : NullReferenceFrame;
	Axis					   : NullAxisRef;
	Station					   : NullStation('Null Station');
	StationCollection		   : NullStationCollection;
	XtsModule				   : NullXtsModule('Null Xts Module');
	XtsModuleCollection		   : NullXtsModuleCollection;
	XtsMover				   : NullXtsMover;
	XtsMoverList			   : NullXtsMoverList;
	XtsMoverData			   : NullXtsMoverData;
	XtsMoverStatus			   : NullXtsMoverStatus;
	XtsMoverTask			   : NullXtsMoverTask;
	XtsMoverTaskCollection	   : NullXtsMoverTaskCollection;
	XtsMoverTaskResult		   : NullXtsMoverTaskResult;
	XtsParameterSet			   : NullXtsParameterSet;
	XtsPart					   : NullXtsPart;
	XtsPartCollection		   : NullXtsPartCollection;
	XtsPositionTrigger		   : NullXtsPositionTrigger;
	XtsPositionTriggerStatus   : NullXtsPositionTriggerStatus;
	XtsStationStatus		   : NullXtsStationStatus;
	XtsTask					   : NullXtsTask;
	XtsTrack				   : NullXtsTrack;
	XtsTrackCollection		   : NullXtsTrackCollection;
	XtsZone					   : NullXtsZone;
	XtsZoneStatus			   : NullXtsZoneStatus;
	ZoneCollection			   : NullZoneCollection;
	SyncAxisParameters		   : NullSyncAxisParameters;
	System					   : NullXtsSystem;
	SystemStatus			   : NullXtsSystemStatus;
	XtsSystemTasks			   : NullXtsSystemTasks;
END_VAR

// Utilities/Logging/XtsTrace
{attribute 'qualified_only'}
VAR_GLOBAL
	{attribute 'hide'}
	EventLogger : XtsCoreEventLogger;
END_VAR

// Version/Global_Version
{attribute 'TcGenerated'}
{attribute 'no-analysis'}
{attribute 'linkalways'}
// This function has been automatically generated from the project information.
VAR_GLOBAL CONSTANT
	{attribute 'const_non_replaced'}
	stLibVersion_XtsCore : ST_LibVersion := (iMajor := 0, iMinor := 12, iBuild := 1, iRevision := 34, nFlags := 0, sVersion := '0.12.1.34');
END_VAR

// XtsCoreParameters
{attribute 'qualified_only'}
VAR_GLOBAL CONSTANT
	InitialTrackId				: UINT	:= 0;
	Nominal24Vdc				: REAL	:= 24.0;
	TcEventLoggerEnabled		: BOOL	:= FALSE;
	MaxNumberLocalLog			: USINT := 20;
	MaxNumberOfMovers			: UDINT := 25;
	MaxNumberOfStations			: UDINT := 10;
	MaxNumberOfPositionTriggers : UDINT := 10;
	MaxNumberOfZones			: UDINT := 10;
	MaxNumberOfParts			: UDINT := 5;
END_VAR

// _Internal/_Needs Sorting/TE2000_Hmi
{attribute 'no_explicit_call' := 'This FB is a CLASS and must be accessed using methods or properties'}
{attribute 'conditionalshow_all_locals'}
{attribute 'hide'}
FUNCTION_BLOCK TE2000_Hmi 
VAR_GENERIC CONSTANT
 	MaxNumberOfMovers : UDINT := 10;
 	MaxNumberOfParts : UDINT := 5;
	MaxNumberOfModules : UDINT := 30;
 	MaxNumberOfStations : UDINT := 5;
 	MaxNumberOfPositionTriggers : UDINT := 5;
 	MaxNumberOfZones : UDINT := 2;
	MaxNumberOfTracks : UDINT := 1;
END_VAR
EXTENDS HmiFunction IMPLEMENTS I_ModuleVisitor, I_ComponentVisitor
VAR
	_System : I_XtsSystem;
	_Parts : ARRAY[1..MaxNumberOfParts] OF ST_XtsPartHmiHelper;
	_PartCount : UINT;
	_ModuleCount : UINT;
	_Movers : XtsMoverCollection;
	_Stations : XtsStationCollection;
	_PositionTriggers : XtsPositionTriggerCollection;
	_Zones : XtsZoneCollection;
	
	{ attribute 'TcHmiSymbol.AddSymbol' }
	{ attribute 'TcHmiSymbol.AddSymbol.UserGroups' := '__SystemAdministrators,Admin' }
	_PartHmiObjects : ARRAY[1..MaxNumberOfParts] OF ST_XtsPart_HMI;
	{ attribute 'TcHmiSymbol.AddSymbol' }
	{ attribute 'TcHmiSymbol.AddSymbol.UserGroups' := '__SystemAdministrators,Admin' }
	_MoverHmiObjects : ARRAY[1..MaxNumberOfMovers] OF ST_XtsMover_HMI;
	{ attribute 'TcHmiSymbol.AddSymbol' }
	{ attribute 'TcHmiSymbol.AddSymbol.UserGroups' := '__SystemAdministrators,Admin' }
	_StationHmiObjects : ARRAY[1..MaxNumberOfStations] OF ST_XtsStation_HMI;
	{ attribute 'TcHmiSymbol.AddSymbol' }
	{ attribute 'TcHmiSymbol.AddSymbol.UserGroups' := '__SystemAdministrators,Admin' }
	_PositionTriggerHmiObjects : ARRAY[1..MaxNumberOfPositionTriggers] OF ST_XtsPositionTrigger_HMI;
	{ attribute 'TcHmiSymbol.AddSymbol' }
	{ attribute 'TcHmiSymbol.AddSymbol.UserGroups' := '__SystemAdministrators,Admin' }
	_ZoneHmiObjects : ARRAY[1..MaxNumberOfZones] OF ST_XtsZone_HMI;
	{ attribute 'TcHmiSymbol.AddSymbol' }
	{ attribute 'TcHmiSymbol.AddSymbol.UserGroups' := '__SystemAdministrators,Admin' }
	_TrackHmiObjects : ARRAY[1..MaxNumberOfTracks] OF ST_XtsTrack_HMI;
	{ attribute 'TcHmiSymbol.AddSymbol' }
	{ attribute 'TcHmiSymbol.AddSymbol.UserGroups' := '__SystemAdministrators,Admin' }
	Xts_HMI : ST_XtsSystem_HMI;
END_VAR

METHOD PRIVATE RefreshXtsModule
VAR_INPUT
	_XtsModule : I_XtsModule;
	HmiModule : POINTER TO ST_XtsModule_Hmi;
END_VAR
HmiModule^.Name		  := _XtsModule.Name;
HmiModule^.Length	  := _XtsModule.Length;
HmiModule^.Gap		  := _XtsModule.Gap;
HmiModule^.CurveAngle := _XtsModule.CurveAngle;
HmiModule^.ModuleType := _XtsModule.XtsModuleType;
END_METHOD

METHOD PRIVATE RefreshXtsMovers
VAR
	_XtsMover : I_XtsMover;
	i		  : UDINT;
END_VAR
_Movers.ResetIterator();
WHILE _Movers.MoveToNext DO
	_XtsMover					 := _Movers.Current;
	i							 := _Movers.CurrentItem;
	_MoverHmiObjects[i].Name	 := _XtsMover.Name;
	_MoverHmiObjects[i].Position := _XtsMover.Position;
END_WHILE
END_METHOD

METHOD PRIVATE RefreshXtsParts
VAR
	_XtsPart   : I_XtsPart;
	i		   : UDINT;
	j		   : UDINT;
	offset	   : ST_OriginTransform;
END_VAR
FOR i := 1 TO TE2000_HMI_Parameters.NUMBER_OF_PARTS DO
	IF _Parts[i].Part = 0 THEN
		//Not a valid part, move on
		EXIT;
	END_IF
	_XtsPart				 := _Parts[i].Part;
	offset					 := _XtsPart.Properties.General.Offset;
	_PartHmiObjects[i].Name	 := _XtsPart.Name;
	_PartHmiObjects[i].Angle := offset.fAlpha;
	_PartHmiObjects[i].X	 := offset.fX;
	_PartHmiObjects[i].Y	 := offset.fY;
	_PartHmiObjects[i].Side	 := _XtsPart.Properties.General.ModuleSide;
	FOR j := 1 TO TE2000_HMI_Parameters.NUMBER_OF_MODULES DO
		IF _Parts[i].Modules[j] = 0 THEN
			//No more modules, exit out
			EXIT;
		END_IF

		RefreshXtsModule(_Parts[i].Modules[j], ADR(_PartHmiObjects[i].Modules[j]));
	END_FOR
END_FOR
END_METHOD

METHOD PRIVATE RefreshXtsPositionTriggers
VAR
	_XtsPositionTrigger : I_XtsPositionTrigger;
	i					: UDINT;
END_VAR
_PositionTriggers.ResetIterator();
WHILE _PositionTriggers.MoveToNext DO
	_XtsPositionTrigger					   := _PositionTriggers.Current;
	i									   := _PositionTriggers.CurrentItem;
	_PositionTriggerHmiObjects[i].Name	   := _XtsPositionTrigger.Name;
	_PositionTriggerHmiObjects[i].Position := _XtsPositionTrigger.Position;
END_WHILE
END_METHOD

METHOD PRIVATE RefreshXtsStations
VAR
	_XtsStation : I_Station;
	i			: UDINT;
END_VAR
_Stations.ResetIterator();
WHILE _Stations.MoveToNext DO
	_XtsStation					   := _Stations.Current;
	i							   := _Stations.CurrentItem;
	_StationHmiObjects[i].Name	   := _XtsStation.Name;
	_StationHmiObjects[i].Position := _XtsStation.Position;
END_WHILE
END_METHOD

METHOD PRIVATE RefreshXtsZones
VAR
	_XtsZone : I_XtsZone;
	i		 : UDINT;
END_VAR
_Zones.ResetIterator();
WHILE _Zones.MoveToNext DO
	_XtsZone						 := _Zones.Current;
	i								 := _Zones.CurrentItem;
	_ZoneHmiObjects[i].Name			 := _XtsZone.Name;
	_ZoneHmiObjects[i].StartPosition := _XtsZone.StartPosition;
	_ZoneHmiObjects[i].EndPosition	 := _XtsZone.EndPosition;
END_WHILE
END_METHOD

METHOD BuildHMI : BOOL
VAR_INPUT
	XtsSystem : I_XtsSystem;
END_VAR
//Reset all the counters and the arrays
MEMSET(ADR(_PartHmiObjects), 0, SIZEOF(_PartHmiObjects));
MEMSET(ADR(_MoverHmiObjects), 0, SIZEOF(_MoverHmiObjects));
MEMSET(ADR(_PositionTriggerHmiObjects), 0, SIZEOF(_PositionTriggerHmiObjects));
MEMSET(ADR(_StationHmiObjects), 0, SIZEOF(_StationHmiObjects));
MEMSET(ADR(_ZoneHmiObjects), 0, SIZEOF(_ZoneHmiObjects));
MEMSET(ADR(_TrackHmiObjects), 0, SIZEOF(_TrackHmiObjects));
MEMSET(ADR(_Parts), 0, SIZEOF(_Parts));
_Movers.Clear();
_Zones.Clear();
_PositionTriggers.Clear();
_Stations.Clear();
_PartCount	 := 0;
_ModuleCount := 0;
_System		 := XtsSystem;
_System.Accept(THIS^);
END_METHOD

PROPERTY ControlObject : I_Base
SET
END_SET
END_PROPERTY

METHOD CyclicLogic
IF _System = 0 THEN
	RETURN;
END_IF
Xts_HMI.Name	  := _System.Name;
Xts_HMI.MoverType := _System.UtilityProperties.Mover.XtsMoverType;
RefreshXtsParts();
RefreshXtsPositionTriggers();
RefreshXtsStations();
RefreshXtsZones();
RefreshXtsMovers();
END_METHOD

(*FB_Init is always available implicitly and it is used primarily for initialization.
The return value is not evaluated. For a specific influence, you can also declare the
methods explicitly and provide additional code there with the standard initialization
code. You can evaluate the return value.*)
METHOD FB_Init : BOOL
VAR_INPUT
	(* TRUE: the retain variables are initialized (reset warm / reset cold)*)
	bInitRetains : BOOL;

	(* TRUE: the instance will be copied to the copy code afterward (online change)   *)
	bInCopyCode : BOOL;
	Name		: Core.T_MaxString;
END_VAR
ControlType := 'XtsSystem';
LinkObject	:= 'Xts_HMI';
END_METHOD

METHOD VisitComponent
VAR_INPUT
	Component : I_Component;
END_VAR

VAR
	_XtsModule			: I_XtsModule;
	_XtsStation			: I_XtsStation;
	_XtsPositionTrigger : I_XtsPositionTrigger;
	_XtsMover			: I_XtsMover;
	_XtsZone			: I_XtsZone;
END_VAR
IF __QUERYINTERFACE(Component, _XtsModule) THEN
	_ModuleCount							 := _ModuleCount + 1;
	_Parts[_PartCount].Modules[_ModuleCount] := _XtsModule;
ELSIF __QUERYINTERFACE(Component, _XtsMover) THEN
	_Movers.AddItem(_XtsMover);
ELSIF __QUERYINTERFACE(Component, _XtsPositionTrigger) THEN
	_PositionTriggers.AddItem(_XtsPositionTrigger);
ELSIF __QUERYINTERFACE(Component, _XtsStation) THEN
	_Stations.AddItem(_XtsStation);
ELSIF __QUERYINTERFACE(Component, _XtsZone) THEN
	_Zones.AddItem(_XtsZone);
END_IF
END_METHOD

METHOD VisitModule
VAR_INPUT
	Module : I_Module;
END_VAR

VAR
	_XtsPart	: I_XtsPart;
END_VAR
IF __QUERYINTERFACE(Module, _XtsPart) THEN
	_PartCount := _PartCount + 1;
	_Parts[_PartCount].Part := _XtsPart;
END_IF

Module.Components.Accept(THIS^);
Module.Modules.Accept(THIS^);
END_METHOD

END_FUNCTION_BLOCK

// XtsSystem/Interfaces/I_XtsSystem
INTERFACE I_XtsSystem EXTENDS I_Module, I_Initializable, I_Cyclic, Core.I_TaskResult, I_XtsXpuId, I_ContainXtsMovers, I_Enablable, I_ContainXtsStations, I_ContainXtsZones, I_ContainXtsTracks,
		I_ContainXtsPositionTriggers, I_HasXtsParameters, I_XtsSystemCommands, I_ContainXtsUtility, I_ContainXtsEnvironment, I_ContainXtsParts, I_ContainXtsSystemProperties,
		I_ContainXtsTracePublisher, I_ContainXtsLocalLog, I_ContainXtsSystemStatus, I_AcceptXtsMoverVisitors, I_AcceptXtsStationVisitor, I_AcceptXtsPositionTriggerVisitor,
		I_AcceptXtsZoneVisitor, I_AcceptXtsPartVisitor, I_AcceptXtsModuleVisitor

{attribute 'monitoring':='call'}
PROPERTY AxesGroupRef : REFERENCE TO AXES_GROUP_REF
GET
END_GET
END_PROPERTY

{attribute 'monitoring':='call'}
PROPERTY Busy : BOOL
GET
END_GET
END_PROPERTY

{attribute 'monitoring' := 'call'}
PROPERTY CAGroupErrorId : UDINT
GET
END_GET
END_PROPERTY

{attribute 'monitoring' := 'call'}
PROPERTY CaGroupStatus : E_MoverGroupState
GET
END_GET
END_PROPERTY

{attribute 'monitoring':='call'}
PROPERTY Config : I_XtsSystemConfiguration
GET
END_GET
END_PROPERTY

{attribute 'monitoring':='call'}
PROPERTY CurrentTask : I_XtsTask
GET
END_GET
END_PROPERTY

{attribute 'monitoring':='call'}
PROPERTY Error : BOOL
GET
END_GET
END_PROPERTY

{attribute 'monitoring':='call'}
PROPERTY ErrorId : UDINT
GET
END_GET
END_PROPERTY

{attribute 'monitoring':='call'}
PROPERTY ManualDiagnoser : REFERENCE TO ManualDebugger
GET
END_GET
END_PROPERTY

{attribute 'monitoring' := 'call'}
PROPERTY MoversEnabled : BOOL
GET
END_GET
END_PROPERTY

PROPERTY XtsTasks : I_XtsTaskCollection
GET
END_GET
END_PROPERTY

END_INTERFACE

// _Internal/TaskBase/Interfaces/I_TaskResult
INTERFACE I_TaskResult EXTENDS Core.I_TaskResult

{attribute 'monitoring':='call'}
PROPERTY TaskName : String
GET
END_GET
END_PROPERTY

END_INTERFACE

// XtsSystem/Interfaces/I_XtsXpuId
INTERFACE I_XtsXpuId EXTENDS I_Base

{attribute 'monitoring':='call'}
PROPERTY XpuId : USINT
GET
END_GET
END_PROPERTY

END_INTERFACE

// XtsSystem/Interfaces/I_ContainXtsMovers
INTERFACE I_ContainXtsMovers EXTENDS I_Base, I_ContainComponents

{attribute 'monitoring':='call'}
PROPERTY Movers : I_XtsMoverCollection
GET
END_GET
END_PROPERTY

END_INTERFACE

// _Internal/Collections/Movers/MoverCollection/Interfaces/I_XtsMoverCollection
INTERFACE I_XtsMoverCollection EXTENDS I_Base, I_XtsMoverEnumerator

METHOD AcceptMoverVisitor
VAR_INPUT
	MoverVisitor : I_XtsMoverVisitor;
END_VAR
END_METHOD

METHOD AddItem
VAR_INPUT
	Mover : I_XtsMover;
END_VAR
END_METHOD

METHOD Clear
VAR_INPUT
END_VAR
END_METHOD

{attribute 'monitoring' := 'call'}
PROPERTY Count : UDINT
GET
END_GET
END_PROPERTY

{attribute 'monitoring' := 'call'}
PROPERTY IsEmpty : BOOL
GET
END_GET
END_PROPERTY

METHOD Remove
VAR_INPUT
	Mover : I_XtsMover;
END_VAR
END_METHOD

END_INTERFACE

// _Internal/Collections/Movers/MoverCollection/Interfaces/I_XtsMoverEnumerator
INTERFACE I_XtsMoverEnumerator EXTENDS I_Base, I_XtsMoverMap, I_AcceptXtsMoverVisitors

{attribute 'monitoring':='call'}
PROPERTY Current : I_XtsMover
GET
END_GET
END_PROPERTY

{attribute 'monitoring' := 'call'}
PROPERTY CurrentItem : UDINT
GET
END_GET
END_PROPERTY

PROPERTY MoveToNext : BOOL
GET
END_GET
END_PROPERTY

METHOD ResetIterator
END_METHOD

END_INTERFACE

// _Internal/Collections/Movers/MoverCollection/Interfaces/I_XtsMoverMap
INTERFACE I_XtsMoverMap EXTENDS I_Base

METHOD Map
VAR_INPUT
	Validator : I_XtsMoverValidator;
	Visitor	  : I_XtsMoverVisitor;
END_VAR
END_METHOD

END_INTERFACE

// XtsMover/Interfaces/I_XtsMoverValidator
INTERFACE I_XtsMoverValidator EXTENDS I_Base

METHOD Valid : BOOL
VAR_INPUT
	Mover : I_XtsMover;
END_VAR
END_METHOD

END_INTERFACE

// XtsMover/Interfaces/I_XtsMover
INTERFACE I_XtsMover EXTENDS I_Component, I_Enablable, I_Resettable, I_Initializable, I_XtsCommands, I_HasXtsParameters, I_AxisRef, I_XtsMoverUtility, I_ContainXtsTracks, I_ContainXtsMoverStatus,
		I_ContainXtsTracePublisher, I_ContainXtsLocalLog, I_AcceptXtsMoverVisitors, I_ContainXtsMoverData, Core.I_TaskResult

{attribute 'monitoring' := 'call'}
PROPERTY CurrentTask : I_XtsMoverTaskResult
GET
END_GET
END_PROPERTY

{attribute 'monitoring' := 'call'}
PROPERTY InPosition : BOOL
GET
END_GET
END_PROPERTY

{attribute 'monitoring':='call'}
PROPERTY InVelocity : BOOL
GET
END_GET
END_PROPERTY

PROPERTY LastCyclePosition : LREAL
GET
END_GET
END_PROPERTY

{attribute 'monitoring':='call'}
PROPERTY ManualGroupControl : BOOL
GET
END_GET
SET
END_SET
END_PROPERTY

{attribute 'monitoring':='call'}
PROPERTY MoverId : UDINT
GET
END_GET
END_PROPERTY

PROPERTY MoverTasks : I_XtsMoverTaskCollection
GET
END_GET
END_PROPERTY

{attribute 'monitoring' := 'call'}
PROPERTY Position : LREAL
GET
END_GET
END_PROPERTY

METHOD RefreshMoverId
VAR_INPUT
	Xpu : I_TcIoXtsProcessingUnit;
END_VAR
END_METHOD

PROPERTY Tracks : I_XtsTrackCollection
GET
END_GET
SET
END_SET
END_PROPERTY

{attribute 'monitoring':='call'}
PROPERTY VirtualMover : BOOL
GET
END_GET
SET
END_SET
END_PROPERTY

END_INTERFACE

// XtsMover/Interfaces/I_XtsCommands
INTERFACE I_XtsCommands EXTENDS I_Base

//Command Mover to Activate to track
METHOD ActivateTrack : I_XtsMoverTaskResult
VAR_INPUT
	TrackId : UDINT; //Track to Activate to
END_VAR
END_METHOD

//Add Mover to CA Group
METHOD AddToGroup : I_XtsMoverTaskResult
VAR_INPUT
	Group : REFERENCE TO AXES_GROUP_REF; //Group to Add to
	Ident : UDINT; //Ident in Group
END_VAR
END_METHOD

//Command Mover to Halt
METHOD Halt : I_XtsMoverTaskResult
VAR_INPUT
	Deceleration : LREAL; //Rate to Decelerate
	Gap			 : LREAL; //Gap to maintain to other movers
END_VAR
END_METHOD

//Command Mover to MoveToPositionRelative
METHOD MoveRelative : I_XtsMoverTaskResult
VAR_INPUT
	Distance  : LREAL; //Distance to move to
END_VAR
END_METHOD

//Command Mover to MoveToPosition
METHOD MoveToPosition : I_XtsMoverTaskResult
VAR_INPUT
	Position	  : LREAL; //Position to move to
	Direction	  : Tc3_Mc3Definitions.MC_DIRECTION := Tc3_Mc3Definitions.MC_DIRECTION.mcDirectionPositive; //Direction to move
END_VAR
END_METHOD

//Command Mover to Move to a Station
METHOD MoveToStation : I_XtsMoverTaskResult
VAR_INPUT
	Station		  : I_XtsStation; //Station to move to
END_VAR
END_METHOD

//Command a Mover to Move At Velocity endlessly
METHOD MoveVelocity : I_XtsMoverTaskResult
VAR_INPUT
	Velocity	  : LREAL; //Velocity to move at
	Direction	  : Tc3_Mc3Definitions.MC_DIRECTION := Tc3_Mc3Definitions.MC_DIRECTION.mcDirectionPositive; //Direction to move
END_VAR
END_METHOD

//Command Mover to remove from CA Group
METHOD RemoveFromGroup : I_XtsMoverTaskResult
VAR_INPUT
	Group : REFERENCE TO AXES_GROUP_REF; //Group to Remvoe Mover From
	Ident : UDINT;                       //Ident of Mover in Group
END_VAR
END_METHOD

//Command Mover to Synchronize to an Axis
METHOD SyncToAxis : I_XtsMoverTaskResult
VAR_INPUT
	Master			   : REFERENCE TO AXIS_REF; //Axis to synchronize to
	MasterSyncPosition : LREAL;					//Master synchronize position					
	SlaveSyncPosition  : LREAL;					//Slave synchronize position
END_VAR
END_METHOD

//Command Mover to Synchronize to another Mover
METHOD SyncToMover : I_XtsMoverTaskResult
VAR_INPUT
	Master	 : I_XtsMover; //Mover to synchronize to
	Distance : LREAL;	   //Distance between movers
END_VAR
END_METHOD

END_INTERFACE

// _Internal/Mover/Tasks/Wrappers/ActivateTrack
FUNCTION_BLOCK ActivateTrack IMPLEMENTS I_ActivateTrack
VAR
	_McActivateTrack : MC_ActivateTrack;
END_VAR

VAR_IN_OUT
	Axis : Tc2_MC2.AXIS_REF;
END_VAR

_McActivateTrack(Axis := Axis);

{attribute 'monitoring':='call'}
PROPERTY Execute : BOOL
GET
Execute := _McActivateTrack.Execute;
END_GET
SET
_McActivateTrack.Execute := Execute;
END_SET
END_PROPERTY

{attribute 'monitoring':='call'}
PROPERTY TrackId : OTCID
GET
TrackId := _McActivateTrack.TrackId;
END_GET
SET
_McActivateTrack.TrackId := TrackId;
END_SET
END_PROPERTY

{attribute 'monitoring':='call'}
PROPERTY Busy : BOOL
GET
Busy := _McActivateTrack.Busy;
END_GET
END_PROPERTY

{attribute 'monitoring':='call'}
PROPERTY Done : BOOL
GET
Done := _McActivateTrack.Done;
END_GET
END_PROPERTY

{attribute 'monitoring':='call'}
PROPERTY Error : BOOL
GET
Error := _McActivateTrack.Error;
END_GET
END_PROPERTY

{attribute 'monitoring':='call'}
PROPERTY ErrorId : UDINT
GET
ErrorId := _McActivateTrack.ErrorId;
END_GET
END_PROPERTY

END_FUNCTION_BLOCK

// _Internal/Mover/Tasks/Wrappers/Interfaces/I_ActivateTrack
INTERFACE I_ActivateTrack EXTENDS I_Base

{attribute 'monitoring':='call'}
PROPERTY Execute : BOOL
GET
END_GET
SET
END_SET
END_PROPERTY

{attribute 'monitoring':='call'}
PROPERTY TrackId : OTCID
GET
END_GET
SET
END_SET
END_PROPERTY

{attribute 'monitoring':='call'}
PROPERTY Busy : BOOL
GET
END_GET
END_PROPERTY

{attribute 'monitoring':='call'}
PROPERTY Error : BOOL
GET
END_GET
END_PROPERTY

{attribute 'monitoring':='call'}
PROPERTY ErrorId : UDINT
GET
END_GET
END_PROPERTY

END_INTERFACE

// _Internal/Mover/MoverTaskBase/Interfaces/I_XtsMoverTaskResult
INTERFACE I_XtsMoverTaskResult EXTENDS I_TaskResult

{attribute 'monitoring':='call'}
PROPERTY Aborted : BOOL
GET
END_GET
END_PROPERTY

PROPERTY CommandExecuted : BOOL
GET
END_GET
END_PROPERTY

{attribute 'monitoring':='call'}
PROPERTY TaskId : MoverTaskId
GET
END_GET
END_PROPERTY

END_INTERFACE

// XtsStation/Interfaces/I_XtsStation
INTERFACE I_XtsStation EXTENDS I_Base, I_Station, I_ContainXtsStationStatus, I_AcceptXtsStationVisitor

END_INTERFACE

// XtsStation/Interfaces/I_Station
INTERFACE I_Station EXTENDS I_Base, I_ContainXtsMoverEnumerator, I_Enablable, I_Positionable, I_Component, I_ContainXtsTracePublisher, I_ContainXtsLocalLog

//Deregisters Mover to be Monitored by Station
METHOD DeregisterMover
VAR_INPUT
	Mover : I_XtsMover; //Mover to Deregister
END_VAR
END_METHOD

//"Gets the Current Mover latched at the Station
METHOD GetMover : I_XtsMover
VAR_INPUT
END_VAR
END_METHOD

//Checks if provided Mover is currently Registered to Station
METHOD IsMoverRegistered : BOOL
VAR_INPUT
	Mover : I_XtsMover; //Mover to check
END_VAR
END_METHOD

{attribute 'monitoring' := 'call'}
PROPERTY MoverIsPresent : BOOL
GET
END_GET
END_PROPERTY

//Registers Mover to be Monitored by Station
METHOD RegisterMover
VAR_INPUT
	Mover : I_XtsMover; //Mover to regsiter
END_VAR
END_METHOD

END_INTERFACE

// _Internal/Collections/I_ContainXtsMoverEnumerator
INTERFACE I_ContainXtsMoverEnumerator EXTENDS I_Base

PROPERTY Movers : I_XtsMoverEnumerator
GET
END_GET
END_PROPERTY

END_INTERFACE

// _Internal/Frames/Interfaces/I_Positionable
INTERFACE I_Positionable EXTENDS I_Base

{attribute 'monitoring' := 'call'}
PROPERTY Position : LREAL
GET
END_GET
SET
END_SET
END_PROPERTY

END_INTERFACE

// Logging/Interfaces/I_ContainXtsTracePublisher
INTERFACE I_ContainXtsTracePublisher EXTENDS I_Base

PROPERTY TracePublisher : I_XtsTracePublisher
GET
END_GET
END_PROPERTY

END_INTERFACE

// Logging/Interfaces/I_XtsTracePublisher
INTERFACE I_XtsTracePublisher EXTENDS I_Base,  I_XtsLogger

METHOD Subscribe
VAR_INPUT
	Logger : I_XtsLogger;
END_VAR
END_METHOD

METHOD Unsubscribe
VAR_INPUT
	Logger : I_XtsLogger;
END_VAR
END_METHOD

END_INTERFACE

// Logging/Interfaces/I_XtsLogger
INTERFACE I_XtsLogger EXTENDS I_TraceLogger, I_TraceInstanceLogger

END_INTERFACE

// Logging/Interfaces/I_ContainXtsLocalLog
INTERFACE I_ContainXtsLocalLog EXTENDS I_Base

{attribute 'monitoring':='call'}
PROPERTY CommandLog : I_XtsLocalLog
GET
END_GET
END_PROPERTY

END_INTERFACE

// Logging/Interfaces/I_XtsLocalLog
INTERFACE I_XtsLocalLog EXTENDS I_Base

METHOD Clear
VAR_INPUT
END_VAR
END_METHOD

{attribute 'monitoring':='call'}
PROPERTY Commands : REFERENCE TO ARRAY[0..XtsCoreParameters.MaxNumberLocalLog - 1] OF T_MaxString
GET
END_GET
END_PROPERTY

{attribute 'monitoring':='call'}
PROPERTY DetailedCommands :  REFERENCE TO ARRAY[0..XtsCoreParameters.MaxNumberLocalLog - 1] OF I_XtsLogCommand
GET
END_GET
END_PROPERTY

END_INTERFACE

// Logging/Interfaces/I_XtsLogCommand
INTERFACE I_XtsLogCommand EXTENDS I_Base, I_TraceMessageInfo, I_TraceSourceInfo, I_ContainTraceArgument

END_INTERFACE

// _Internal/Station/Status/Interfaces/I_ContainXtsStationStatus
INTERFACE I_ContainXtsStationStatus EXTENDS I_Base

{attribute 'monitoring':='call'}
PROPERTY Status : I_XtsStationStatus
GET
END_GET
END_PROPERTY

END_INTERFACE

// _Internal/Station/Status/Interfaces/I_XtsStationStatus
INTERFACE I_XtsStationStatus EXTENDS I_Base

{attribute 'monitoring':='call'}
//Number of Movers Currently Registered to the Station
PROPERTY NumberOfMoversRegistered : UDINT
GET
END_GET
END_PROPERTY

END_INTERFACE

// XtsStation/Interfaces/I_AcceptXtsStationVisitor
INTERFACE I_AcceptXtsStationVisitor EXTENDS I_Base

METHOD AcceptStationVisitor
VAR_INPUT
	StationVisitor : I_XtsStationVisitor;
END_VAR
END_METHOD

END_INTERFACE

// XtsStation/Interfaces/I_XtsStationVisitor
INTERFACE I_XtsStationVisitor EXTENDS I_Base

METHOD VisitStation
VAR_INPUT
	Station : I_Station;
END_VAR
END_METHOD

END_INTERFACE

// _Internal/Mover/Parameters/Interfaces/I_HasXtsParameters
INTERFACE I_HasXtsParameters EXTENDS I_Base

{attribute 'monitoring' := 'call'}
PROPERTY Parameters : I_XtsParameterSet
GET
END_GET
SET
END_SET
END_PROPERTY

END_INTERFACE

// _Internal/Mover/Parameters/Interfaces/I_XtsParameterSet
INTERFACE I_XtsParameterSet EXTENDS I_Base, I_BaseDynamics, I_CollisionAvoidanceDynamics, I_MoveToPositionParameters, I_XtsTrackParameter, I_ContainSyncAxisParameters

METHOD CopyFrom
VAR_INPUT
	Other : I_XtsParameterSet;
END_VAR
END_METHOD

METHOD CopyTo
VAR_INPUT
	Other : I_XtsParameterSet;
END_VAR
END_METHOD

END_INTERFACE

// _Internal/Mover/Parameters/Interfaces/I_BaseDynamics
INTERFACE I_BaseDynamics EXTENDS I_Base

{attribute 'monitoring':='call'}
PROPERTY Acceleration : LREAL
GET
END_GET
SET
END_SET
END_PROPERTY

{attribute 'monitoring':='call'}
PROPERTY Deceleration : LREAL
GET
END_GET
SET
END_SET
END_PROPERTY

{attribute 'monitoring':='call'}
PROPERTY Direction : Tc3_Mc3Definitions.MC_DIRECTION;
GET
END_GET
SET
END_SET
END_PROPERTY

{attribute 'monitoring' := 'call'}
PROPERTY Jerk : LREAL
GET
END_GET
SET
END_SET
END_PROPERTY

{attribute 'monitoring':='call'}
PROPERTY Velocity : LREAL
GET
END_GET
SET
END_SET
END_PROPERTY

END_INTERFACE

// _Internal/Mover/Parameters/Interfaces/I_CollisionAvoidanceDynamics
INTERFACE I_CollisionAvoidanceDynamics EXTENDS I_Base

{attribute 'monitoring':='call'}
PROPERTY Gap : LREAL
GET
END_GET
SET
END_SET
END_PROPERTY

END_INTERFACE

// _Internal/Mover/Parameters/Interfaces/I_MoveToPositionParameters
INTERFACE I_MoveToPositionParameters EXTENDS I_Base

{attribute 'monitoring' := 'call'}
PROPERTY Position : LREAL
GET
END_GET
SET
END_SET
END_PROPERTY

END_INTERFACE

// _Internal/Mover/Parameters/Interfaces/I_XtsTrackParameter
INTERFACE I_XtsTrackParameter EXTENDS I_Base

{attribute 'monitoring' := 'call'}
PROPERTY Track : I_XtsTrack
GET
END_GET
SET
END_SET
END_PROPERTY

END_INTERFACE

// _Internal/Tracks/Interfaces/I_XtsTrack
INTERFACE I_XtsTrack EXTENDS I_Base, I_Disposable

{attribute 'monitoring':='call'}
PROPERTY Id : UDINT
GET
END_GET
SET
END_SET
END_PROPERTY

{attribute 'monitoring':='call'}
PROPERTY Length : LREAL
GET
END_GET
SET
END_SET
END_PROPERTY

{attribute 'monitoring':='call'}
PROPERTY Offset : LREAL
GET
END_GET
SET
END_SET
END_PROPERTY

{attribute 'monitoring':='call'}
PROPERTY Otcid : OTCID
GET
END_GET
SET
END_SET
END_PROPERTY

{attribute 'monitoring':='call'}
PROPERTY Polarity : Polarity
GET
END_GET
SET
END_SET
END_PROPERTY

PROPERTY Utility : I_TcIoXtsXpuTrack
GET
END_GET
SET
END_SET
END_PROPERTY

END_INTERFACE

// _Internal/Mover/Parameters/Interfaces/I_ContainSyncAxisParameters
INTERFACE I_ContainSyncAxisParameters EXTENDS I_Base

{attribute 'monitoring':='call'}
PROPERTY SyncAxis : I_SyncAxisParameters
GET
END_GET
END_PROPERTY

END_INTERFACE

// _Internal/Mover/Parameters/Interfaces/I_SyncAxisParameters
INTERFACE I_SyncAxisParameters EXTENDS I_Base

{attribute 'monitoring':='call'}
PROPERTY MasterAxis : REFERENCE TO AXIS_REF
GET
END_GET
SET
END_SET
END_PROPERTY

{attribute 'monitoring' := 'call'}
PROPERTY MasterStartDistance : MC_LREAL
GET
END_GET
SET
END_SET
END_PROPERTY

{attribute 'monitoring' := 'call'}
PROPERTY MasterSyncPosition : MC_LREAL
GET
END_GET
SET
END_SET
END_PROPERTY

PROPERTY Options_CA : REFERENCE TO Tc3_McCollisionAvoidance.ST_GearInPosCAOptions
GET
END_GET
SET
END_SET
END_PROPERTY

{attribute 'monitoring' := 'call'}
PROPERTY RatioDenominator : UINT
GET
END_GET
SET
END_SET
END_PROPERTY

{attribute 'monitoring' := 'call'}
PROPERTY RatioNumerator : MC_LREAL
GET
END_GET
SET
END_SET
END_PROPERTY

{attribute 'monitoring' := 'call'}
PROPERTY SlaveSyncPosition : LREAL
GET
END_GET
SET
END_SET
END_PROPERTY

{attribute 'monitoring' := 'call'}
PROPERTY SyncMode : Tc3_McCollisionAvoidance.MC_SYNC_MODE
GET
END_GET
SET
END_SET
END_PROPERTY

{attribute 'monitoring' := 'call'}
PROPERTY SyncStrategy : Tc3_McCollisionAvoidance.MC_SYNC_STRATEGY
GET
END_GET
SET
END_SET
END_PROPERTY

END_INTERFACE

// _Internal/Mover/Tasks/Interfaces/I_AxisRef
INTERFACE I_AxisRef EXTENDS I_Base

PROPERTY Axis : REFERENCE TO Tc2_MC2.AXIS_REF
GET
END_GET
END_PROPERTY

END_INTERFACE

// XtsMover/Interfaces/I_XtsMoverUtility
INTERFACE I_XtsMoverUtility EXTENDS I_Base

PROPERTY MoverUtility : I_TcIoXtsXpuMover
GET
END_GET
SET
END_SET
END_PROPERTY

END_INTERFACE

// XtsSystem/Interfaces/I_ContainXtsTracks
INTERFACE I_ContainXtsTracks EXTENDS I_Base

PROPERTY Tracks : I_XtsTrackCollection
GET
END_GET
END_PROPERTY

END_INTERFACE

// _Internal/Collections/Tracks/TrackCollection/Interfaces/I_XtsTrackCollection
INTERFACE I_XtsTrackCollection EXTENDS I_Base, I_XtsTrackEnumerator

METHOD Clear
VAR_INPUT
END_VAR
END_METHOD

{attribute 'monitoring' := 'call'}
PROPERTY Count : UDINT
GET
END_GET
END_PROPERTY

{attribute 'hide'}
METHOD Create : BOOL
VAR_INPUT
	NumberOfTracks : UINT;
END_VAR
END_METHOD

METHOD GetById : I_XtsTrack
VAR_INPUT
	TrackId : UDINT;
END_VAR
END_METHOD

METHOD GetByOtcid : I_XtsTrack
VAR_INPUT
	TrackOtcid : OTCID;
END_VAR
END_METHOD

{attribute 'monitoring' := 'call'}
PROPERTY IsEmpty : BOOL
GET
END_GET
END_PROPERTY

END_INTERFACE

// _Internal/Collections/Tracks/TrackCollection/Interfaces/I_XtsTrackEnumerator
INTERFACE I_XtsTrackEnumerator EXTENDS I_Base

{attribute 'monitoring':='call'}
PROPERTY Current : I_XtsTrack
GET
END_GET
END_PROPERTY

{attribute 'monitoring' := 'call'}
PROPERTY CurrentIndex : UDINT
GET
END_GET
END_PROPERTY

PROPERTY MoveToNext : BOOL
GET
END_GET
END_PROPERTY

METHOD ResetIterator
END_METHOD

END_INTERFACE

// _Internal/Mover/Status/Interfaces/I_ContainXtsMoverStatus
INTERFACE I_ContainXtsMoverStatus EXTENDS I_Base

{attribute 'monitoring':='call'}
PROPERTY Status : I_XtsMoverStatus
GET
END_GET
END_PROPERTY

END_INTERFACE

// _Internal/Mover/Status/Interfaces/I_XtsMoverStatus
INTERFACE I_XtsMoverStatus EXTENDS I_Base

{attribute 'monitoring':='call'}
PROPERTY ActualAcceleration : LREAL
GET
END_GET
END_PROPERTY

{attribute 'monitoring':='call'}
PROPERTY ActualVelocity : LREAL
GET
END_GET
END_PROPERTY

{attribute 'monitoring':='call'}
PROPERTY AvoidingCollision : BOOL
GET
END_GET
END_PROPERTY

{attribute 'monitoring':='call'}
PROPERTY Axis : I_AxisRef
GET
END_GET
END_PROPERTY

{attribute 'monitoring':='call'}
PROPERTY CommandedPosition : LREAL
GET
END_GET
SET
END_SET
END_PROPERTY

{attribute 'monitoring':='call'}
PROPERTY CommandedStation : I_XtsStation
GET
END_GET
SET
END_SET
END_PROPERTY

{attribute 'monitoring':='call'}
PROPERTY CurrentTrack : I_XtsTrack
GET
END_GET
SET
END_SET
END_PROPERTY

{attribute 'monitoring':='call'}
PROPERTY IdentInGroup : UDINT
GET
END_GET
SET
END_SET
END_PROPERTY

{attribute 'monitoring' := 'call'}
PROPERTY InSync : BOOL
GET
END_GET
SET
END_SET
END_PROPERTY

{attribute 'monitoring':='call'}
PROPERTY MoverInGroup : BOOL
GET
END_GET
END_PROPERTY

{attribute 'monitoring':='call'}
PROPERTY SetAcceleration : LREAL
GET
END_GET
END_PROPERTY

{attribute 'monitoring':='call'}
PROPERTY SetVelocity : LREAL
GET
END_GET
END_PROPERTY

END_INTERFACE

// XtsMover/Interfaces/I_AcceptXtsMoverVisitors
INTERFACE I_AcceptXtsMoverVisitors EXTENDS I_Base

METHOD AcceptMoverVisitor
VAR_INPUT
	MoverVisitor : I_XtsMoverVisitor;
END_VAR
END_METHOD

END_INTERFACE

// XtsMover/Interfaces/I_XtsMoverVisitor
INTERFACE I_XtsMoverVisitor EXTENDS I_Base

METHOD VisitMover
VAR_INPUT
	Mover : I_XtsMover;
END_VAR
END_METHOD

END_INTERFACE

// XtsMover/XtsMoverData/Interfaces/I_ContainXtsMoverData
INTERFACE I_ContainXtsMoverData EXTENDS I_Base

{attribute 'monitoring':='call'}
PROPERTY MoverData : I_XtsMoverData
GET
END_GET
SET
END_SET
END_PROPERTY

END_INTERFACE

// XtsMover/XtsMoverData/Interfaces/I_XtsMoverData
INTERFACE I_XtsMoverData EXTENDS I_Base

END_INTERFACE

// _Internal/Mover/MoverTaskBase/Interfaces/I_XtsMoverTaskCollection
INTERFACE I_XtsMoverTaskCollection

METHOD AddTask : BOOL
VAR_INPUT
	Task   : I_XtsMoverTask;
END_VAR
END_METHOD

PROPERTY ErrorTask : T_MaxString
GET
END_GET
END_PROPERTY

METHOD GetTaskById : I_XtsMoverTask
VAR_INPUT
	TaskId : MoverTaskID;
END_VAR
END_METHOD

METHOD GetTaskByName : I_XtsMoverTask
VAR_INPUT
	Name : T_MaxString;
END_VAR
END_METHOD

METHOD RemoveTaskById : BOOL
VAR_INPUT
	TaskId : MoverTaskId;
END_VAR
END_METHOD

METHOD RemoveTaskByInstance : BOOL
VAR_INPUT
	Task : I_XtsMoverTask;
END_VAR
END_METHOD

END_INTERFACE

// _Internal/Mover/MoverTaskBase/Interfaces/I_XtsMoverTask
INTERFACE I_XtsMoverTask EXTENDS I_Base, I_XtsMoverTaskResult, I_Cyclic, I_Resettable

PROPERTY Axis : I_AxisRef
GET
END_GET
SET
END_SET
END_PROPERTY

METHOD Execute : I_XtsMoverTaskResult
VAR_INPUT
END_VAR
END_METHOD

END_INTERFACE

// XtsSystem/Interfaces/I_ContainXtsStations
INTERFACE I_ContainXtsStations EXTENDS I_Base, I_ContainComponents

PROPERTY Stations : I_XtsStationCollection
GET
END_GET
END_PROPERTY

END_INTERFACE

// _Internal/Collections/Stations/StationCollection/Interfaces/I_XtsStationCollection
INTERFACE I_XtsStationCollection EXTENDS I_Base,I_XtsStationEnumerator

METHOD AddItem
VAR_INPUT
	Station : I_XtsStation;
END_VAR
END_METHOD

METHOD Clear
VAR_INPUT
END_VAR
END_METHOD

{attribute 'monitoring' := 'call'}
PROPERTY Count : UDINT
GET
END_GET
END_PROPERTY

{attribute 'monitoring' := 'call'}
PROPERTY IsEmpty : BOOL
GET
END_GET
END_PROPERTY

METHOD Remove
VAR_INPUT
	Station : I_XtsStation;
END_VAR
END_METHOD

END_INTERFACE

// _Internal/Collections/Stations/StationCollection/Interfaces/I_XtsStationEnumerator
INTERFACE I_XtsStationEnumerator EXTENDS I_Base, I_AcceptXtsStationVisitor

{attribute 'monitoring':='call'}
PROPERTY Current : I_XtsStation
GET
END_GET
END_PROPERTY

{attribute 'monitoring' := 'call'}
PROPERTY CurrentItem : UDINT
GET
END_GET
END_PROPERTY

PROPERTY MoveToNext : BOOL
GET
END_GET
END_PROPERTY

METHOD ResetIterator
END_METHOD

END_INTERFACE

// XtsSystem/Interfaces/I_ContainXtsZones
INTERFACE I_ContainXtsZones EXTENDS I_Base, I_ContainComponents

PROPERTY Zones : I_XtsZoneCollection
GET
END_GET
END_PROPERTY

END_INTERFACE

// _Internal/Collections/Zones/ZoneCollection/Interfaces/I_XtsZoneCollection
INTERFACE I_XtsZoneCollection EXTENDS I_Base,I_XtsZoneEnumerator

METHOD AddItem
VAR_INPUT
	Zone : I_XtsZone;
END_VAR
END_METHOD

METHOD Clear
VAR_INPUT
END_VAR
END_METHOD

{attribute 'monitoring' := 'call'}
PROPERTY Count : UDINT
GET
END_GET
END_PROPERTY

{attribute 'monitoring' := 'call'}
PROPERTY IsEmpty : BOOL
GET
END_GET
END_PROPERTY

METHOD Remove
VAR_INPUT
	Zone : I_XtsZone;
END_VAR
END_METHOD

END_INTERFACE

// _Internal/Collections/Zones/ZoneCollection/Interfaces/I_XtsZoneEnumerator
INTERFACE I_XtsZoneEnumerator EXTENDS I_Base

{attribute 'monitoring':='call'}
PROPERTY Current : I_XtsZone
GET
END_GET
END_PROPERTY

{attribute 'monitoring' := 'call'}
PROPERTY CurrentItem : UDINT
GET
END_GET
END_PROPERTY

PROPERTY MoveToNext : BOOL
GET
END_GET
END_PROPERTY

METHOD ResetIterator
END_METHOD

END_INTERFACE

// XtsZone/Interfaces/I_XtsZone
INTERFACE I_XtsZone EXTENDS I_Base, I_Component, I_ContainXtsMoverEnumerator, I_MonitorsMovers, I_SingleDimensionZone, I_ContainXtsZoneStatus, I_ContainXtsTracePublisher,
		I_ContainXtsLocalLog, I_AcceptXtsMoverVisitors, I_AcceptXtsZoneVisitor

//Select the Nth Mover in the Zone
METHOD GetSortedMover : I_XtsMover
VAR_INPUT
	Index	  : UDINT; // 1 based index
	Direction : Tc3_Mc3Definitions.MC_DIRECTION := Tc3_Mc3Definitions.MC_DIRECTION.mcDirectionPositive; //Direction to fetch from
END_VAR
END_METHOD

METHOD IsMoverInZone : BOOL
VAR_INPUT
	Mover : I_XtsMover;
END_VAR
END_METHOD

END_INTERFACE

// XtsZone/Interfaces/I_MonitorsMovers
INTERFACE I_MonitorsMovers EXTENDS I_Base

PROPERTY MonitoredMovers : I_XtsMoverCollection
SET
END_SET
END_PROPERTY

END_INTERFACE

// _Internal/Zone/Properties/Interfaces/I_SingleDimensionZone
INTERFACE I_SingleDimensionZone EXTENDS I_Base

{attribute 'monitoring' := 'call'}
PROPERTY EndPosition : LREAL
GET
END_GET
SET
END_SET
END_PROPERTY

{attribute 'monitoring' := 'call'}
PROPERTY StartPosition : LREAL
GET
END_GET
SET
END_SET
END_PROPERTY

END_INTERFACE

// _Internal/Zone/Status/Interfaces/I_ContainXtsZoneStatus
INTERFACE I_ContainXtsZoneStatus EXTENDS I_Base

{attribute 'monitoring':='call'}
PROPERTY Status : I_XtsZoneStatus
GET
END_GET
END_PROPERTY

END_INTERFACE

// _Internal/Zone/Status/Interfaces/I_XtsZoneStatus
INTERFACE I_XtsZoneStatus EXTENDS I_Base

{attribute 'monitoring':='call'}
//Number of Movers Currently in Zone
PROPERTY NumberOfMoversInZone : UDINT
GET
END_GET
END_PROPERTY

END_INTERFACE

// XtsZone/Interfaces/I_AcceptXtsZoneVisitor
INTERFACE I_AcceptXtsZoneVisitor EXTENDS I_Base

METHOD AcceptXtsZoneVisitor
VAR_INPUT
	ZoneVisitor : I_XtsZoneVisitor;
END_VAR
END_METHOD

END_INTERFACE

// XtsZone/Interfaces/I_XtsZoneVisitor
INTERFACE I_XtsZoneVisitor EXTENDS I_Base

METHOD VisitZone
VAR_INPUT
	Zone : I_XtsZone;
END_VAR
END_METHOD

END_INTERFACE

// XtsSystem/Interfaces/I_ContainXtsPositionTriggers
INTERFACE I_ContainXtsPositionTriggers EXTENDS I_Base, I_ContainComponents

PROPERTY PositionTriggers : I_XtsPositionTriggerCollection
GET
END_GET
END_PROPERTY

END_INTERFACE

// _Internal/Collections/PositionTriggers/PositionTriggerCollection/Interfaces/I_XtsPositionTriggerCollection
INTERFACE I_XtsPositionTriggerCollection EXTENDS I_Base,I_XtsPositionTriggerEnumerator

METHOD AddItem
VAR_INPUT
	PositionTrigger : I_XtsPositionTrigger;
END_VAR
END_METHOD

METHOD Clear
VAR_INPUT
END_VAR
END_METHOD

{attribute 'monitoring' := 'call'}
PROPERTY Count : UDINT
GET
END_GET
END_PROPERTY

{attribute 'monitoring' := 'call'}
PROPERTY IsEmpty : BOOL
GET
END_GET
END_PROPERTY

METHOD Remove
VAR_INPUT
	PositionTrigger : I_XtsPositionTrigger;
END_VAR
END_METHOD

END_INTERFACE

// _Internal/Collections/PositionTriggers/PositionTriggerCollection/Interfaces/I_XtsPositionTriggerEnumerator
INTERFACE I_XtsPositionTriggerEnumerator EXTENDS I_Base, I_AcceptXtsPositionTriggerVisitor

{attribute 'monitoring':='call'}
PROPERTY Current : I_XtsPositionTrigger
GET
END_GET
END_PROPERTY

{attribute 'monitoring' := 'call'}
PROPERTY CurrentItem : UDINT
GET
END_GET
END_PROPERTY

PROPERTY MoveToNext : BOOL
GET
END_GET
END_PROPERTY

METHOD ResetIterator
END_METHOD

END_INTERFACE

// XtsPositionTrigger/Interfaces/I_AcceptXtsPositionTriggerVisitor
INTERFACE I_AcceptXtsPositionTriggerVisitor EXTENDS I_Base

METHOD AcceptXtsPositionTriggerVisitor
VAR_INPUT
	PositionTriggerVisitor : I_VisitXtsPositionTrigger;
END_VAR
END_METHOD

END_INTERFACE

// XtsPositionTrigger/Interfaces/I_VisitXtsPositionTrigger
INTERFACE I_VisitXtsPositionTrigger EXTENDS I_Base

METHOD VisitXtsPositionTrigger
VAR_INPUT
	PositionTrigger : I_XtsPositionTrigger;
END_VAR
END_METHOD

END_INTERFACE

// XtsPositionTrigger/Interfaces/I_XtsPositionTrigger
INTERFACE I_XtsPositionTrigger EXTENDS I_Station, I_Positionable, I_Queueable, I_AcceptXtsPositionTriggerVisitor, I_ContainXtsPositionTriggerStatus

PROPERTY Movers : I_XtsMoverEnumerator
GET
END_GET
SET
END_SET
END_PROPERTY

END_INTERFACE

// XtsPositionTrigger/Interfaces/I_Queueable
INTERFACE I_Queueable EXTENDS I_Base

{attribute 'monitoring':='call'}
PROPERTY MoverQueue : I_XtsMoverQueue
GET
END_GET
END_PROPERTY

END_INTERFACE

// _Internal/Collections/Movers/MoverQueue/Interfaces/I_XtsMoverQueue
INTERFACE I_XtsMoverQueue EXTENDS I_Base, I_XtsMoverEnumerator

METHOD Clear
VAR_INPUT
END_VAR
END_METHOD

{attribute 'monitoring':='call'}
PROPERTY Count : UDINT
GET
END_GET
END_PROPERTY

METHOD Dequeue : I_XtsMover
END_METHOD

METHOD Enqueue
VAR_INPUT
	Mover : I_XtsMover;
END_VAR
END_METHOD

METHOD Peek : I_XtsMover
END_METHOD

END_INTERFACE

// _Internal/PositionTrigger/Status/Interfaces/I_ContainXtsPositionTriggerStatus
INTERFACE I_ContainXtsPositionTriggerStatus EXTENDS I_Base

{attribute 'monitoring':='call'}
PROPERTY Status : I_XtsPositionTriggerStatus
GET
END_GET
END_PROPERTY

END_INTERFACE

// _Internal/PositionTrigger/Status/Interfaces/I_XtsPositionTriggerStatus
INTERFACE I_XtsPositionTriggerStatus EXTENDS I_Base

{attribute 'monitoring':='call'}
//Number of Movers that have occurred and are in the current queue
PROPERTY NumberOfMoverEvents : UDINT
GET
END_GET
END_PROPERTY

{attribute 'monitoring':='call'}
//Number of Movers Currently Registered to the PositionTrigger
PROPERTY NumberOfMoversRegistered : UDINT
GET
END_GET
END_PROPERTY

END_INTERFACE

// XtsSystem/Interfaces/I_XtsSystemCommands
INTERFACE I_XtsSystemCommands EXTENDS I_Base, I_Resettable

METHOD DisableGroup
VAR_INPUT
END_VAR
END_METHOD

METHOD DisableMovers
VAR_INPUT
END_VAR
END_METHOD

METHOD EnableGroup
VAR_INPUT
END_VAR
END_METHOD

METHOD EnableMovers
VAR_INPUT
END_VAR
END_METHOD

METHOD ResetCaGroup
VAR_INPUT
END_VAR
END_METHOD

METHOD ResetMovers
VAR_INPUT
END_VAR
END_METHOD

METHOD RetriggerMoverDetection
VAR_INPUT
END_VAR
END_METHOD

METHOD TriggerMoverDetection
VAR_INPUT
END_VAR
END_METHOD

METHOD TriggerMoverIdentification
VAR_INPUT
END_VAR
END_METHOD

END_INTERFACE

// XtsSystem/Interfaces/I_ContainXtsUtility
INTERFACE I_ContainXtsUtility EXTENDS I_Base

PROPERTY Utility : I_TcIoXtsProcessingUnit
GET
END_GET
SET
END_SET
END_PROPERTY

END_INTERFACE

// XtsSystem/Interfaces/I_ContainXtsEnvironment
INTERFACE I_ContainXtsEnvironment EXTENDS I_Base

PROPERTY Environment : I_TcIoXtsEnvironment
GET
END_GET
SET
END_SET
END_PROPERTY

END_INTERFACE

// _Internal/Collections/Parts/PartCollection/Interfaces/I_ContainXtsParts
INTERFACE I_ContainXtsParts EXTENDS I_Base

PROPERTY Parts : I_XtsPartCollection
GET
END_GET
END_PROPERTY

END_INTERFACE

// _Internal/Collections/Parts/PartCollection/Interfaces/I_XtsPartCollection
INTERFACE I_XtsPartCollection EXTENDS I_Base, I_XtsPartEnumerator

METHOD AddItem
VAR_INPUT
	Part : I_XtsPart;
END_VAR
END_METHOD

METHOD Clear
VAR_INPUT
END_VAR
END_METHOD

{attribute 'monitoring' := 'call'}
PROPERTY Count : UDINT
GET
END_GET
END_PROPERTY

METHOD GetById : I_XtsPart
VAR_INPUT
	PartId : UDINT;
END_VAR
END_METHOD

METHOD GetByOtcid : I_XtsPart
VAR_INPUT
	PartOtcid : OTCID;
END_VAR
END_METHOD

{attribute 'monitoring' := 'call'}
PROPERTY IsEmpty : BOOL
GET
END_GET
END_PROPERTY

METHOD Remove
VAR_INPUT
	Part : I_XtsPart;
END_VAR
END_METHOD

END_INTERFACE

// _Internal/Collections/Parts/PartCollection/Interfaces/I_XtsPartEnumerator
INTERFACE I_XtsPartEnumerator EXTENDS I_Base

{attribute 'monitoring':='call'}
PROPERTY Current : I_XtsPart
GET
END_GET
END_PROPERTY

{attribute 'monitoring' := 'call'}
PROPERTY CurrentItem : UDINT
GET
END_GET
END_PROPERTY

PROPERTY MoveToNext : BOOL
GET
END_GET
END_PROPERTY

METHOD ResetIterator
END_METHOD

END_INTERFACE

// XtsPart/Interfaces/I_XtsPart
INTERFACE I_XtsPart
	EXTENDS I_Base, I_Module, I_Initializable, I_XtsPartId, I_ContainXtsPartUtility, I_ContainXtsModules, I_Disposable, I_ContainXtsPartProperties, I_AcceptXtsPartVisitor, I_AcceptXtsModuleVisitor

PROPERTY PartReady : BOOL
GET
END_GET
END_PROPERTY

{attribute 'monitoring':='call'}
//Combined Vdc24Okay for All Modules
PROPERTY Vdc24Okay : BOOL
GET
END_GET
END_PROPERTY

{attribute 'monitoring':='call'}
//Combined Vdc48Okay for All Modules
PROPERTY Vdc48Okay : BOOL
GET
END_GET
END_PROPERTY

END_INTERFACE

// _Internal/Parts/I_XtsPartId
INTERFACE I_XtsPartId EXTENDS I_Base

PROPERTY XtsPartId : UINT
GET
END_GET
SET
END_SET
END_PROPERTY

END_INTERFACE

// XtsPart/Interfaces/I_ContainXtsPartUtility
INTERFACE I_ContainXtsPartUtility EXTENDS I_Base

{attribute 'monitoring':='call'}
PROPERTY Utility : I_TcIoXtsXpuPart
GET
END_GET
SET
END_SET
END_PROPERTY

END_INTERFACE

// _Internal/Collections/Modules/ModuleCollection/Interfaces/I_ContainXtsModules
INTERFACE I_ContainXtsModules EXTENDS I_Base

{attribute 'monitoring':='call'}
PROPERTY XtsModules : I_XtsModuleCollection
GET
END_GET
END_PROPERTY

END_INTERFACE

// _Internal/Collections/Modules/ModuleCollection/Interfaces/I_XtsModuleCollection
INTERFACE I_XtsModuleCollection EXTENDS I_Base, I_XtsModuleEnumerator, I_Disposable

METHOD Clear
VAR_INPUT
END_VAR
END_METHOD

{attribute 'monitoring' := 'call'}
PROPERTY Count : UDINT
GET
END_GET
END_PROPERTY

{attribute 'hide'}
METHOD Create : BOOL
VAR_INPUT
	NumberOfModules : UINT;
END_VAR
END_METHOD

METHOD GetById : I_XtsModule
VAR_INPUT
	ModuleId : UDINT;
END_VAR
END_METHOD

METHOD GetByOtcid : I_XtsModule
VAR_INPUT
	ModuleOtcid : OTCID;
END_VAR
END_METHOD

{attribute 'monitoring' := 'call'}
PROPERTY IsEmpty : BOOL
GET
END_GET
END_PROPERTY

END_INTERFACE

// _Internal/Collections/Modules/ModuleCollection/Interfaces/I_XtsModuleEnumerator
INTERFACE I_XtsModuleEnumerator EXTENDS I_Base

{attribute 'monitoring':='call'}
PROPERTY Current : I_XtsModule
GET
END_GET
END_PROPERTY

{attribute 'monitoring' := 'call'}
PROPERTY CurrentItem : UDINT
GET
END_GET
END_PROPERTY

PROPERTY MoveToNext : BOOL
GET
END_GET
END_PROPERTY

METHOD ResetIterator
END_METHOD

END_INTERFACE

// XtsModule/Interfaces/I_XtsModule
INTERFACE I_XtsModule EXTENDS I_Component, I_Disposable, I_ContainXtsPartModuleUtility, I_Initializable, I_AcceptXtsModuleVisitor

{attribute 'monitoring':='call'}
PROPERTY CurveAngle : LREAL
GET
END_GET
END_PROPERTY

{attribute 'monitoring':='call'}
PROPERTY Gap : LREAL
GET
END_GET
END_PROPERTY

{attribute 'monitoring':='call'}
PROPERTY Id : UDINT
GET
END_GET
SET
END_SET
END_PROPERTY

{attribute 'monitoring':='call'}
PROPERTY Length : LREAL
GET
END_GET
END_PROPERTY

{attribute 'monitoring':='call'}
PROPERTY ModuleReady : BOOL
GET
END_GET
END_PROPERTY

{attribute 'monitoring':='call'}
PROPERTY Otcid : OTCID
GET
END_GET
SET
END_SET
END_PROPERTY

{attribute 'monitoring':='call'}
PROPERTY Vdc24Okay : BOOL
GET
END_GET
END_PROPERTY

{attribute 'monitoring':='call'}
PROPERTY Vdc48Okay : BOOL
GET
END_GET
END_PROPERTY

{attribute 'monitoring':='call'}
PROPERTY XtsModuleType : Tc3_Xts_Utility.ModuleType
GET
END_GET
END_PROPERTY

END_INTERFACE

// XtsModule/Interfaces/I_ContainXtsPartModuleUtility
INTERFACE I_ContainXtsPartModuleUtility EXTENDS I_Base

{attribute 'monitoring':='call'}
PROPERTY Utility : I_TcIoXtsPartModule
GET
END_GET
SET
END_SET
END_PROPERTY

END_INTERFACE

// XtsModule/Interfaces/I_AcceptXtsModuleVisitor
INTERFACE I_AcceptXtsModuleVisitor EXTENDS I_Base

METHOD AcceptXtsModuleVisitor
VAR_INPUT
	XtsModuleVisitor : I_XtsModuleVisitor;
END_VAR
END_METHOD

END_INTERFACE

// XtsModule/Interfaces/I_XtsModuleVisitor
INTERFACE I_XtsModuleVisitor EXTENDS I_Base

METHOD VisitXtsModule
VAR_INPUT
	XtsModule : I_XtsModule;
END_VAR
END_METHOD

END_INTERFACE

// XtsModule/XtsModule
{attribute 'no_explicit_call' := 'This FB is a CLASS and must be accessed using methods or properties'}
{attribute 'hide_all_locals'}
{attribute 'enable_dynamic_creation'}
FUNCTION_BLOCK XtsModule EXTENDS CyclicComponent IMPLEMENTS I_XtsModule
VAR
	_Simulated	 : BOOL;
	_Otcid		 : OTCID;
	_Id			 : UDINT;
	_Utility	 : I_TcIoXtsPartModule;
	_Module24Vdc : REAL;
	_Module48Vdc : REAL;
	_Initialized : BOOL;
	_Length		 : LREAL;
	_ModuleGap	 : LREAL;
	_CurveAngle	 : LREAL;
	_ModuleType	 : Tc3_XTS_Utility.ModuleType;
	_ModuleReady : BOOL;
END_VAR

METHOD DeregisterWithParent
VAR_INPUT
	Parent	: Core.I_ContainComponents;
END_VAR
Parent.DeregisterInitialize(THIS^);
SUPER^.DeregisterWithParent(Parent);
END_METHOD

METHOD RegisterWithParent
VAR_INPUT
	Parent	: Core.I_ContainComponents;
END_VAR
Parent.RegisterInitialize(THIS^);
SUPER^.RegisterWithParent(Parent);
END_METHOD

METHOD Dispose
VAR
	pDispose : POINTER TO XtsModule;
END_VAR
pDispose := THIS;
__DELETE(pDispose);
END_METHOD

METHOD Initialize
IF _Utility = 0 THEN
	RETURN;
END_IF

_Name		 := CONCAT('Module ', UDINT_TO_STRING(_Utility.GetGlobalNumber()));
_Length		 := _Utility.GetLength();
_ModuleGap	 := _Utility.GetGap();
_CurveAngle	 := _Utility.GetAngle();
_ModuleType	 := _Utility.GetModuleType();
_Initialized := TRUE;
END_METHOD

{attribute 'monitoring' := 'call'}
PROPERTY Initialized : BOOL
GET
Initialized := _Initialized;
END_GET
SET
_Initialized := Initialized;
END_SET
END_PROPERTY

{attribute 'monitoring':='call'}
PROPERTY CurveAngle : LREAL
GET
CurveAngle := _CurveAngle;
END_GET
END_PROPERTY

{attribute 'monitoring':='call'}
PROPERTY Gap : LREAL
GET
Gap := _ModuleGap;
END_GET
END_PROPERTY

{attribute 'monitoring':='call'}
PROPERTY Id : UDINT
GET
Id := _Id;
END_GET
SET
_Id := Id;
END_SET
END_PROPERTY

{attribute 'monitoring':='call'}
PROPERTY Length : LREAL
GET
Length := _Length;
END_GET
END_PROPERTY

{attribute 'monitoring':='call'}
PROPERTY ModuleReady : BOOL
GET
ModuleReady := _ModuleReady;
END_GET
END_PROPERTY

{attribute 'monitoring':='call'}
PROPERTY Otcid : OTCID
GET
Otcid := _Otcid;
END_GET
SET
_Otcid := Otcid;
END_SET
END_PROPERTY

{attribute 'monitoring':='call'}
PROPERTY Utility : I_TcIoXtsPartModule
GET
Utility := _Utility;
END_GET
SET
_Utility := Utility;
END_SET
END_PROPERTY

{attribute 'monitoring':='call'}
PROPERTY Vdc24Okay : BOOL
GET
Vdc24Okay := _Module24Vdc > (XtsCoreParameters.Nominal24Vdc * 0.9) AND _Module24Vdc < (XtsCoreParameters.Nominal24Vdc * 1.1);
END_GET
END_PROPERTY

{attribute 'monitoring':='call'}
PROPERTY Vdc48Okay : BOOL
GET
Vdc48Okay := _Utility.GetIsDcLinkVoltageReady();
END_GET
END_PROPERTY

{attribute 'monitoring':='call'}
PROPERTY XtsModuleType : Tc3_Xts_Utility.ModuleType
GET
XtsModuleType := _ModuleType;
END_GET
END_PROPERTY

METHOD AcceptXtsModuleVisitor
VAR_INPUT
	XtsModuleVisitor : I_XtsModuleVisitor;
END_VAR
XtsModuleVisitor.VisitXtsModule(THIS^);
END_METHOD

METHOD CyclicLogic
IF _Simulated OR _Utility = 0 THEN
	RETURN;
END_IF

_Module24Vdc := _Utility.GetAuxiliaryVoltage24V();
IF Vdc24Okay AND Vdc48Okay THEN
	_ModuleReady := TRUE;
ELSE
	_ModuleReady := FALSE;
END_IF
END_METHOD

END_FUNCTION_BLOCK

// _Internal/Parts/Properties/I_ContainXtsPartProperties
INTERFACE I_ContainXtsPartProperties EXTENDS I_Base

PROPERTY Properties : I_XtsPartProperties
GET
END_GET
END_PROPERTY

END_INTERFACE

// _Internal/Parts/Properties/I_XtsPartProperties
INTERFACE I_XtsPartProperties EXTENDS I_Base

PROPERTY General : I_XtsPartPropertiesGeneral
GET
END_GET
END_PROPERTY

END_INTERFACE

// _Internal/Parts/Properties/I_XtsPartPropertiesGeneral
INTERFACE I_XtsPartPropertiesGeneral EXTENDS I_Base

PROPERTY ModuleSide : Tc3_Xts_Utility.ModuleSide
GET
END_GET
SET
END_SET
END_PROPERTY

PROPERTY Offset : ST_OriginTransform
GET
END_GET
SET
END_SET
END_PROPERTY

PROPERTY OTCID : OTCID
GET
END_GET
SET
END_SET
END_PROPERTY

END_INTERFACE

// XtsPart/Interfaces/I_AcceptXtsPartVisitor
INTERFACE I_AcceptXtsPartVisitor EXTENDS I_Base

METHOD AcceptXtsPartVisitor
VAR_INPUT
	XtsPartVisitor : I_XtsPartVisitor;
END_VAR
END_METHOD

END_INTERFACE

// XtsPart/Interfaces/I_XtsPartVisitor
INTERFACE I_XtsPartVisitor EXTENDS I_Base

METHOD VisitXtsPart
VAR_INPUT
	XtsPart : I_XtsPart;
END_VAR
END_METHOD

END_INTERFACE

// XtsPart/XtsPart
{attribute 'no_explicit_call' := 'This FB is a CLASS and must be accessed using methods or properties'}
{attribute 'enable_dynamic_creation'}
FUNCTION_BLOCK XtsPart EXTENDS Module IMPLEMENTS I_XtsPart
VAR
	_Simulated : BOOL;
	_Otcid	   : OTCID;
	_Id		   : UINT;
	_Utility   : I_TcIoXtsXpuPart;
	{attribute 'hide'}
	_Properties : XtsPartProperties;
	_ModuleReadyCount : UINT;
	_ModuleNotReadyCount :UINT;

	//
	_DefaultInitializeTask : InitializeXtsPartTask;
	_InitializeTask		   : I_XtsPartInitializeTask := _DefaultInitializeTask;

	// 
	_ModuleCollection : XtsModuleCollection;
END_VAR

//FB_Init is always available implicitly and it is used primarily for initialization.

//The return value is not evaluated. For a specific influence, you can also declare the

//methods explicitly and provide additional code there with the standard initialization

//code. You can evaluate the return value.
METHOD FB_Init : BOOL
VAR_INPUT
	bInitRetains : BOOL;		// TRUE: the retain variables are initialized (reset warm / reset cold)
	bInCopyCode	 : BOOL;		// TRUE: the instance will be copied to the copy code afterward (online change)
	Name		 : T_MaxString; //Name of the XtsPart
END_VAR
_InitializeTask.XtsPartId := THIS^;
END_METHOD

METHOD Dispose
VAR
	pDispose : POINTER TO XtsPart;
END_VAR
pDispose := THIS;

_ModuleCollection.Clear();
__DELETE(pDispose);
END_METHOD

(* This Module will be done initialize when ModuleInitialized := TRUE;, subequently all subitems will be called to be initialized *)
METHOD Initializing
_InitializeTask.Initialize();
IF NOT _InitializeTask.Busy THEN
	_Name := CONCAT('Part ', UDINT_TO_STRING(_Utility.GetGlobalNumber()));
END_IF

ModuleInitialized := NOT _InitializeTask.Busy AND NOT _InitializeTask.Error;
END_METHOD

PROPERTY Properties : I_XtsPartProperties
GET
Properties := _Properties;
END_GET
END_PROPERTY

PROPERTY PartReady : BOOL
GET
PartReady := Vdc24Okay AND Vdc48Okay;
END_GET
END_PROPERTY

{attribute 'monitoring':='call'}
//Combined Vdc24Okay for All Modules
PROPERTY Vdc24Okay : BOOL
GET
VAR
	VoltageOk : BOOL;
END_VAR
VoltageOk := TRUE;
_ModuleCollection.ResetIterator();
WHILE _ModuleCollection.MoveToNext DO
	VoltageOk := VoltageOk AND _ModuleCollection.Current.Vdc24Okay;
END_WHILE
Vdc24Okay := VoltageOk;
END_GET
END_PROPERTY

{attribute 'monitoring':='call'}
//Combined Vdc48Okay for All Modules
PROPERTY Vdc48Okay : BOOL
GET
Vdc48Okay := _Utility.GetIsDcLinkVoltageReady();
END_GET
END_PROPERTY

METHOD AcceptXtsModuleVisitor
VAR_INPUT
	XtsModuleVisitor : I_XtsModuleVisitor;
END_VAR
_ModuleCollection.ResetIterator();
WHILE _ModuleCollection.MoveToNext DO
	_ModuleCollection.Current.AcceptXtsModuleVisitor(XtsModuleVisitor);
END_WHILE
END_METHOD

METHOD AcceptXtsPartVisitor
VAR_INPUT
	XtsPartVisitor : I_XtsPartVisitor;
END_VAR
XtsPartVisitor.VisitXtsPart(THIS^);
END_METHOD

METHOD OnCyclicCall
VAR
	Module : I_XtsModule;
END_VAR
IF _Utility = 0 THEN
	RETURN;
END_IF

RETURN;

_ModuleReadyCount	 := 0;
_ModuleNotReadyCount := 0;
_ModuleCollection.ResetIterator();
WHILE _ModuleCollection.MoveToNext DO
	Module	   := _ModuleCollection.Current;
	IF Module.ModuleReady THEN
		_ModuleReadyCount := _ModuleReadyCount + 1;
	ELSE
		_ModuleNotReadyCount := _ModuleNotReadyCount + 1;
	END_IF
END_WHILE
END_METHOD

{attribute 'monitoring':='call'}
PROPERTY Utility : I_TcIoXtsXpuPart
GET
Utility := _Utility;
END_GET
SET
_Utility := Utility;
END_SET
END_PROPERTY

{attribute 'monitoring':='call'}
//Collection of XtsModules assigned to Part
PROPERTY XtsModules : I_XtsModuleCollection
GET
XtsModules := _ModuleCollection;
END_GET
END_PROPERTY

PROPERTY XtsPartId : UINT
GET
XtsPartId := _Id;
END_GET
SET
_Id := XtsPartId;
END_SET
END_PROPERTY

END_FUNCTION_BLOCK

// _Internal/Parts/Properties/XtsPartProperties
{attribute 'no_explicit_call' := 'This FB is a CLASS and must be accessed using methods or properties'}
{attribute 'hide_all_locals'}
FUNCTION_BLOCK XtsPartProperties IMPLEMENTS I_XtsPartProperties
VAR
	_General : XtsPartPropertiesGeneral;
END_VAR

PROPERTY General : I_XtsPartPropertiesGeneral
GET
General := _General;
END_GET
END_PROPERTY

END_FUNCTION_BLOCK

